gfCNCPoint3[9678] = {X 502.6885, Y 49.3200, Z -3.8333, A 0.000, B 0.000, C 0.000 }
gfCNCPoint3[9679] = {X 496.2450, Y 49.3200, Z -3.8333, A 0.000, B 0.000, C 0.000 }
gfCNCPoint3[9680] = {X 495.2885, Y 49.2128, Z -3.8333, A 0.000, B 0.000, C 0.000 }
gfCNCPoint3[9681] = {X 494.3794, Y 48.8964, Z -3.8333, A 0.000, B 0.000, C 0.000 }
gfCNCPoint3[9682] = {X 493.5630, Y 48.3866, Z -3.8333, A 0.000, B 0.000, C 0.000 }
gfCNCPoint3[9683] = {X 492.8797, Y 47.7087, Z -3.8333, A 0.000, B 0.000, C 0.000 }
gfCNCPoint3[9684] = {X 492.3635, Y 46.8963, Z -3.8333, A 0.000, B 0.000, C 0.000 }
gfCNCPoint3[9685] = {X 492.0399, Y 45.9898, Z -3.8333, A 0.000, B 0.000, C 0.000 }
gfCNCPoint3[9686] = {X 491.9252, Y 45.0341, Z -3.8333, A 0.000, B 0.000, C 0.000 }
gfCNCPoint3[9687] = {X 491.9254, Y 44.1494, Z -3.8333, A 0.000, B 0.000, C 0.000 }
gfCNCPoint3[9688] = {X 492.0359, Y 43.2364, Z -3.8333, A 0.000, B 0.000, C 0.000 }
gfCNCPoint3[9689] = {X 492.3371, Y 42.3675, Z -3.8333, A 0.000, B 0.000, C 0.000 }
gfCNCPoint3[9690] = {X 492.8153, Y 41.5821, Z -3.8333, A 0.000, B 0.000, C 0.000 }
gfCNCPoint3[9691] = {X 493.4490, Y 40.9157, Z -3.8333, A 0.000, B 0.000, C 0.000 }
gfCNCPoint3[9692] = {X 493.4490, Y 34.4738, Z -3.8333, A 0.000, B 0.000, C 0.000 }
gfCNCPoint3[9693] = {X 490.7241, Y 34.4738, Z -3.8333, A 0.000, B 0.000, C 0.000 }
gfCNCPoint3[9694] = {X 486.4400, Y 42.8164, Z -3.8333, A 0.000, B 0.000, C 0.000 }
gfCNCPoint3[9695] = {X 486.4449, Y 42.8296, Z -3.8333, A 0.000, B 0.000, C 0.000 }
gfCNCPoint3[9696] = {X 486.6109, Y 43.4908, Z -3.8333, A 0.000, B 0.000, C 0.000 }
gfCNCPoint3[9697] = {X 486.6708, Y 44.1699, Z -3.8333, A 0.000, B 0.000, C 0.000 }
gfCNCPoint3[9698] = {X 486.6710, Y 45.0000, Z -3.8333, A 0.000, B 0.000, C 0.000 }
gfCNCPoint3[9699] = {X 486.5627, Y 45.9613, Z -3.8333, A 0.000, B 0.000, C 0.000 }
gfCNCPoint3[9700] = {X 486.2432, Y 46.8744, Z -3.8333, A 0.000, B 0.000, C 0.000 }
gfCNCPoint3[9701] = {X 485.7285, Y 47.6935, Z -3.8333, A 0.000, B 0.000, C 0.000 }
gfCNCPoint3[9702] = {X 485.0445, Y 48.3775, Z -3.8333, A 0.000, B 0.000, C 0.000 }
gfCNCPoint3[9703] = {X 484.2254, Y 48.8922, Z -3.8333, A 0.000, B 0.000, C 0.000 }
gfCNCPoint3[9704] = {X 483.3123, Y 49.2117, Z -3.8333, A 0.000, B 0.000, C 0.000 }
gfCNCPoint3[9705] = {X 482.3510, Y 49.3200, Z -3.8333, A 0.000, B 0.000, C 0.000 }
gfCNCPoint3[9706] = {X 475.7650, Y 49.3200, Z -3.8333, A 0.000, B 0.000, C 0.000 }
gfCNCPoint3[9707] = {X 474.8037, Y 49.2117, Z -3.8333, A 0.000, B 0.000, C 0.000 }
gfCNCPoint3[9708] = {X 473.8906, Y 48.8922, Z -3.8333, A 0.000, B 0.000, C 0.000 }
gfCNCPoint3[9709] = {X 473.0715, Y 48.3775, Z -3.8333, A 0.000, B 0.000, C 0.000 }
gfCNCPoint3[9710] = {X 472.3875, Y 47.6935, Z -3.8333, A 0.000, B 0.000, C 0.000 }
gfCNCPoint3[9711] = {X 471.8728, Y 46.8745, Z -3.8333, A 0.000, B 0.000, C 0.000 }
gfCNCPoint3[9712] = {X 471.5533, Y 45.9614, Z -3.8333, A 0.000, B 0.000, C 0.000 }
gfCNCPoint3[9713] = {X 471.4450, Y 45.0001, Z -3.8333, A 0.000, B 0.000, C 0.000 }
gfCNCPoint3[9714] = {X 471.4454, Y 44.1494, Z -3.8333, A 0.000, B 0.000, C 0.000 }
gfCNCPoint3[9715] = {X 471.5430, Y 43.2935, Z -3.8333, A 0.000, B 0.000, C 0.000 }
gfCNCPoint3[9716] = {X 471.8086, Y 42.4740, Z -3.8333, A 0.000, B 0.000, C 0.000 }
gfCNCPoint3[9717] = {X 472.2314, Y 41.7236, Z -3.8333, A 0.000, B 0.000, C 0.000 }
gfCNCPoint3[9718] = {X 472.7947, Y 41.0719, Z -3.8333, A 0.000, B 0.000, C 0.000 }
gfCNCPoint3[9719] = {X 473.4762, Y 40.5449, Z -3.8333, A 0.000, B 0.000, C 0.000 }
gfCNCPoint3[9720] = {X 474.2486, Y 40.1637, Z -3.8333, A 0.000, B 0.000, C 0.000 }
gfCNCPoint3[9721] = {X 478.2331, Y 32.3645, Z -3.8333, A 0.000, B 0.000, C 0.000 }
gfCNCPoint3[9722] = {X 476.9697, Y 31.4968, Z -3.8333, A 0.000, B 0.000, C 0.000 }
gfCNCPoint3[9723] = {X 475.8333, Y 30.4684, Z -3.8333, A 0.000, B 0.000, C 0.000 }
gfCNCPoint3[9724] = {X 474.8441, Y 29.2977, Z -3.8333, A 0.000, B 0.000, C 0.000 }
gfCNCPoint3[9725] = {X 474.0198, Y 28.0056, Z -3.8333, A 0.000, B 0.000, C 0.000 }
gfCNCPoint3[9726] = {X 473.3752, Y 26.6150, Z -3.8333, A 0.000, B 0.000, C 0.000 }
gfCNCPoint3[9727] = {X 472.9218, Y 25.1510, Z -3.8333, A 0.000, B 0.000, C 0.000 }
gfCNCPoint3[9728] = {X 472.6083, Y 23.4679, Z -3.8333, A 0.000, B 0.000, C 0.000 }
gfCNCPoint3[9729] = {X 472.4682, Y 21.7616, Z -3.8333, A 0.000, B 0.000, C 0.000 }
gfCNCPoint3[9730] = {X 472.5029, Y 20.0499, Z -3.8333, A 0.000, B 0.000, C 0.000 }
gfCNCPoint3[9731] = {X 472.7121, Y 18.3506, Z -3.8333, A 0.000, B 0.000, C 0.000 }
gfCNCPoint3[9732] = {X 473.0935, Y 16.6816, Z -3.8333, A 0.000, B 0.000, C 0.000 }
gfCNCPoint3[9733] = {X 473.6361, Y 15.1667, Z -3.8333, A 0.000, B 0.000, C 0.000 }
gfCNCPoint3[9734] = {X 474.3793, Y 13.7395, Z -3.8333, A 0.000, B 0.000, C 0.000 }
gfCNCPoint3[9735] = {X 475.3094, Y 12.4264, Z -3.8333, A 0.000, B 0.000, C 0.000 }
gfCNCPoint3[9736] = {X 476.4090, Y 11.2517, Z -3.8333, A 0.000, B 0.000, C 0.000 }
gfCNCPoint3[9737] = {X 477.6579, Y 10.2370, Z -3.8333, A 0.000, B 0.000, C 0.000 }
gfCNCPoint3[9738] = {X 479.0330, Y 9.4012, Z -3.8333, A 0.000, B 0.000, C 0.000 }
gfCNCPoint3[9739] = {X 480.5087, Y 8.7598, Z -3.8333, A 0.000, B 0.000, C 0.000 }
gfCNCPoint3[9740] = {X 482.0579, Y 8.3246, Z -3.8333, A 0.000, B 0.000, C 0.000 }
gfCNCPoint3[9741] = {X 484.1552, Y 7.9976, Z -3.8333, A 0.000, B 0.000, C 0.000 }
gfCNCPoint3[9742] = {X 486.2747, Y 7.8831, Z -3.8333, A 0.000, B 0.000, C 0.000 }
gfCNCPoint3[9743] = {X 486.9679, Y 7.8709, Z -3.8333, A 0.000, B 0.000, C 0.000 }
gfCNCPoint3[9744] = {X 492.3835, Y 7.8709, Z -3.8333, A 0.000, B 0.000, C 0.000 }
gfCNCPoint3[9745] = {X 492.3835, Y 3.8709, Z -3.8333, A 0.000, B 0.000, C 0.000 }
gfCNCPoint3[9746] = {X 492.3835, Y 7.9509, Z -3.8333, A 0.000, B 0.000, C 0.000 }
gfCNCPoint3[9747] = {X 502.2063, Y 7.9509, Z -3.8333, A 0.000, B 0.000, C 0.000 }
gfCNCPoint3[9748] = {X 502.7388, Y 7.9551, Z -3.8333, A 0.000, B 0.000, C 0.000 }
gfCNCPoint3[9749] = {X 503.6730, Y 8.0672, Z -3.8333, A 0.000, B 0.000, C 0.000 }
gfCNCPoint3[9750] = {X 504.5591, Y 8.3834, Z -3.8333, A 0.000, B 0.000, C 0.000 }
gfCNCPoint3[9751] = {X 505.3533, Y 8.8880, Z -3.8333, A 0.000, B 0.000, C 0.000 }
gfCNCPoint3[9752] = {X 506.0160, Y 9.5559, Z -3.8333, A 0.000, B 0.000, C 0.000 }
gfCNCPoint3[9753] = {X 506.5144, Y 10.3540, Z -3.8333, A 0.000, B 0.000, C 0.000 }
gfCNCPoint3[9754] = {X 506.8237, Y 11.2426, Z -3.8333, A 0.000, B 0.000, C 0.000 }
gfCNCPoint3[9755] = {X 506.9285, Y 12.1776, Z -3.8333, A 0.000, B 0.000, C 0.000 }
gfCNCPoint3[9756] = {X 506.9285, Y 12.9781, Z -3.8333, A 0.000, B 0.000, C 0.000 }
gfCNCPoint3[9757] = {X 506.8270, Y 13.9000, Z -3.8333, A 0.000, B 0.000, C 0.000 }
gfCNCPoint3[9758] = {X 506.5276, Y 14.7777, Z -3.8333, A 0.000, B 0.000, C 0.000 }
gfCNCPoint3[9759] = {X 506.0445, Y 15.5693, Z -3.8333, A 0.000, B 0.000, C 0.000 }
gfCNCPoint3[9760] = {X 505.4009, Y 16.2369, Z -3.8333, A 0.000, B 0.000, C 0.000 }
gfCNCPoint3[9761] = {X 505.4008, Y 40.9504, Z -3.8333, A 0.000, B 0.000, C 0.000 }
gfCNCPoint3[9762] = {X 505.4291, Y 40.9736, Z -3.8333, A 0.000, B 0.000, C 0.000 }
gfCNCPoint3[9763] = {X 506.0558, Y 41.6322, Z -3.8333, A 0.000, B 0.000, C 0.000 }
gfCNCPoint3[9764] = {X 506.5277, Y 42.4092, Z -3.8333, A 0.000, B 0.000, C 0.000 }
gfCNCPoint3[9765] = {X 506.8230, Y 43.2690, Z -3.8333, A 0.000, B 0.000, C 0.000 }
gfCNCPoint3[9766] = {X 506.9283, Y 44.1720, Z -3.8333, A 0.000, B 0.000, C 0.000 }
gfCNCPoint3[9767] = {X 506.9285, Y 45.0000, Z -3.8333, A 0.000, B 0.000, C 0.000 }
gfCNCPoint3[9768] = {X 506.8222, Y 45.9435, Z -3.8333, A 0.000, B 0.000, C 0.000 }
gfCNCPoint3[9769] = {X 506.5086, Y 46.8397, Z -3.8333, A 0.000, B 0.000, C 0.000 }
gfCNCPoint3[9770] = {X 506.0035, Y 47.6436, Z -3.8333, A 0.000, B 0.000, C 0.000 }
gfCNCPoint3[9771] = {X 505.3321, Y 48.3150, Z -3.8333, A 0.000, B 0.000, C 0.000 }
gfCNCPoint3[9772] = {X 504.5282, Y 48.8201, Z -3.8333, A 0.000, B 0.000, C 0.000 }
gfCNCPoint3[9773] = {X 503.6320, Y 49.1337, Z -3.8333, A 0.000, B 0.000, C 0.000 }
gfCNCPoint3[9774] = {X 502.6885, Y 49.2400, Z -3.8333, A 0.000, B 0.000, C 0.000 }
gfCNCPoint3[9775] = {X 496.2450, Y 49.2400, Z -3.8333, A 0.000, B 0.000, C 0.000 }
gfCNCPoint3[9776] = {X 495.3062, Y 49.1348, Z -3.8333, A 0.000, B 0.000, C 0.000 }
gfCNCPoint3[9777] = {X 494.4140, Y 48.8242, Z -3.8333, A 0.000, B 0.000, C 0.000 }
gfCNCPoint3[9778] = {X 493.6127, Y 48.3239, Z -3.8333, A 0.000, B 0.000, C 0.000 }
gfCNCPoint3[9779] = {X 492.9420, Y 47.6585, Z -3.8333, A 0.000, B 0.000, C 0.000 }
gfCNCPoint3[9780] = {X 492.4354, Y 46.8612, Z -3.8333, A 0.000, B 0.000, C 0.000 }
gfCNCPoint3[9781] = {X 492.1178, Y 45.9714, Z -3.8333, A 0.000, B 0.000, C 0.000 }
gfCNCPoint3[9782] = {X 492.0052, Y 45.0335, Z -3.8333, A 0.000, B 0.000, C 0.000 }
gfCNCPoint3[9783] = {X 492.0054, Y 44.1505, Z -3.8333, A 0.000, B 0.000, C 0.000 }
gfCNCPoint3[9784] = {X 492.1159, Y 43.2454, Z -3.8333, A 0.000, B 0.000, C 0.000 }
gfCNCPoint3[9785] = {X 492.4173, Y 42.3850, Z -3.8333, A 0.000, B 0.000, C 0.000 }
gfCNCPoint3[9786] = {X 492.8957, Y 41.6088, Z -3.8333, A 0.000, B 0.000, C 0.000 }
gfCNCPoint3[9787] = {X 493.5290, Y 40.9529, Z -3.8333, A 0.000, B 0.000, C 0.000 }
gfCNCPoint3[9788] = {X 493.5290, Y 34.3938, Z -3.8333, A 0.000, B 0.000, C 0.000 }
gfCNCPoint3[9789] = {X 490.6753, Y 34.3938, Z -3.8333, A 0.000, B 0.000, C 0.000 }
gfCNCPoint3[9790] = {X 486.3526, Y 42.8115, Z -3.8333, A 0.000, B 0.000, C 0.000 }
gfCNCPoint3[9791] = {X 486.3696, Y 42.8564, Z -3.8333, A 0.000, B 0.000, C 0.000 }
gfCNCPoint3[9792] = {X 486.5322, Y 43.5048, Z -3.8333, A 0.000, B 0.000, C 0.000 }
gfCNCPoint3[9793] = {X 486.5908, Y 44.1706, Z -3.8333, A 0.000, B 0.000, C 0.000 }
gfCNCPoint3[9794] = {X 486.5910, Y 45.0000, Z -3.8333, A 0.000, B 0.000, C 0.000 }
gfCNCPoint3[9795] = {X 486.4847, Y 45.9435, Z -3.8333, A 0.000, B 0.000, C 0.000 }
gfCNCPoint3[9796] = {X 486.1711, Y 46.8397, Z -3.8333, A 0.000, B 0.000, C 0.000 }
gfCNCPoint3[9797] = {X 485.6660, Y 47.6436, Z -3.8333, A 0.000, B 0.000, C 0.000 }
gfCNCPoint3[9798] = {X 484.9946, Y 48.3150, Z -3.8333, A 0.000, B 0.000, C 0.000 }
gfCNCPoint3[9799] = {X 484.1907, Y 48.8201, Z -3.8333, A 0.000, B 0.000, C 0.000 }
gfCNCPoint3[9800] = {X 483.2945, Y 49.1337, Z -3.8333, A 0.000, B 0.000, C 0.000 }
gfCNCPoint3[9801] = {X 482.3510, Y 49.2400, Z -3.8333, A 0.000, B 0.000, C 0.000 }
gfCNCPoint3[9802] = {X 475.7650, Y 49.2400, Z -3.8333, A 0.000, B 0.000, C 0.000 }
gfCNCPoint3[9803] = {X 474.8215, Y 49.1337, Z -3.8333, A 0.000, B 0.000, C 0.000 }
gfCNCPoint3[9804] = {X 473.9253, Y 48.8201, Z -3.8333, A 0.000, B 0.000, C 0.000 }
gfCNCPoint3[9805] = {X 473.1214, Y 48.3150, Z -3.8333, A 0.000, B 0.000, C 0.000 }
gfCNCPoint3[9806] = {X 472.4500, Y 47.6436, Z -3.8333, A 0.000, B 0.000, C 0.000 }
gfCNCPoint3[9807] = {X 471.9449, Y 46.8397, Z -3.8333, A 0.000, B 0.000, C 0.000 }
gfCNCPoint3[9808] = {X 471.6313, Y 45.9436, Z -3.8333, A 0.000, B 0.000, C 0.000 }
gfCNCPoint3[9809] = {X 471.5250, Y 45.0001, Z -3.8333, A 0.000, B 0.000, C 0.000 }
gfCNCPoint3[9810] = {X 471.5254, Y 44.1505, Z -3.8333, A 0.000, B 0.000, C 0.000 }
gfCNCPoint3[9811] = {X 471.6223, Y 43.3054, Z -3.8333, A 0.000, B 0.000, C 0.000 }
gfCNCPoint3[9812] = {X 471.8860, Y 42.4967, Z -3.8333, A 0.000, B 0.000, C 0.000 }
gfCNCPoint3[9813] = {X 472.3057, Y 41.7570, Z -3.8333, A 0.000, B 0.000, C 0.000 }
gfCNCPoint3[9814] = {X 472.8647, Y 41.1159, Z -3.8333, A 0.000, B 0.000, C 0.000 }
gfCNCPoint3[9815] = {X 473.5404, Y 40.5992, Z -3.8333, A 0.000, B 0.000, C 0.000 }
gfCNCPoint3[9816] = {X 474.3057, Y 40.2278, Z -3.8333, A 0.000, B 0.000, C 0.000 }
gfCNCPoint3[9817] = {X 478.3386, Y 32.3338, Z -3.8333, A 0.000, B 0.000, C 0.000 }
gfCNCPoint3[9818] = {X 477.0685, Y 31.4727, Z -3.8333, A 0.000, B 0.000, C 0.000 }
gfCNCPoint3[9819] = {X 475.9257, Y 30.4488, Z -3.8333, A 0.000, B 0.000, C 0.000 }
gfCNCPoint3[9820] = {X 474.9308, Y 29.2805, Z -3.8333, A 0.000, B 0.000, C 0.000 }
gfCNCPoint3[9821] = {X 474.1021, Y 27.9891, Z -3.8333, A 0.000, B 0.000, C 0.000 }
gfCNCPoint3[9822] = {X 473.4544, Y 26.5980, Z -3.8333, A 0.000, B 0.000, C 0.000 }
gfCNCPoint3[9823] = {X 472.9996, Y 25.1325, Z -3.8333, A 0.000, B 0.000, C 0.000 }
gfCNCPoint3[9824] = {X 472.6876, Y 23.4574, Z -3.8333, A 0.000, B 0.000, C 0.000 }
gfCNCPoint3[9825] = {X 472.5482, Y 21.7592, Z -3.8333, A 0.000, B 0.000, C 0.000 }
gfCNCPoint3[9826] = {X 472.5827, Y 20.0556, Z -3.8333, A 0.000, B 0.000, C 0.000 }
gfCNCPoint3[9827] = {X 472.7909, Y 18.3645, Z -3.8333, A 0.000, B 0.000, C 0.000 }
gfCNCPoint3[9828] = {X 473.1704, Y 16.7034, Z -3.8333, A 0.000, B 0.000, C 0.000 }
gfCNCPoint3[9829] = {X 473.7094, Y 15.1988, Z -3.8333, A 0.000, B 0.000, C 0.000 }
gfCNCPoint3[9830] = {X 474.4476, Y 13.7812, Z -3.8333, A 0.000, B 0.000, C 0.000 }
gfCNCPoint3[9831] = {X 475.3714, Y 12.4770, Z -3.8333, A 0.000, B 0.000, C 0.000 }
gfCNCPoint3[9832] = {X 476.4636, Y 11.3102, Z -3.8333, A 0.000, B 0.000, C 0.000 }
gfCNCPoint3[9833] = {X 477.7040, Y 10.3024, Z -3.8333, A 0.000, B 0.000, C 0.000 }
gfCNCPoint3[9834] = {X 479.0698, Y 9.4722, Z -3.8333, A 0.000, B 0.000, C 0.000 }
gfCNCPoint3[9835] = {X 480.5356, Y 8.8351, Z -3.8333, A 0.000, B 0.000, C 0.000 }
gfCNCPoint3[9836] = {X 482.0742, Y 8.4029, Z -3.8333, A 0.000, B 0.000, C 0.000 }
gfCNCPoint3[9837] = {X 484.1638, Y 8.0772, Z -3.8333, A 0.000, B 0.000, C 0.000 }
gfCNCPoint3[9838] = {X 486.2756, Y 7.9631, Z -3.8333, A 0.000, B 0.000, C 0.000 }
gfCNCPoint3[9839] = {X 486.9686, Y 7.9509, Z -3.8333, A 0.000, B 0.000, C 0.000 }
gfCNCPoint3[9840] = {X 492.3835, Y 7.9509, Z -3.8333, A 0.000, B 0.000, C 0.000 }
gfCNCPoint3[9841] = {X 492.3835, Y 3.9509, Z -3.8333, A 0.000, B 0.000, C 0.000 }
gfCNCPoint3[9842] = {X 492.3835, Y 8.0309, Z -3.8333, A 0.000, B 0.000, C 0.000 }
gfCNCPoint3[9843] = {X 502.2059, Y 8.0309, Z -3.8333, A 0.000, B 0.000, C 0.000 }
gfCNCPoint3[9844] = {X 502.7381, Y 8.0351, Z -3.8333, A 0.000, B 0.000, C 0.000 }
gfCNCPoint3[9845] = {X 503.6546, Y 8.1451, Z -3.8333, A 0.000, B 0.000, C 0.000 }
gfCNCPoint3[9846] = {X 504.5240, Y 8.4553, Z -3.8333, A 0.000, B 0.000, C 0.000 }
gfCNCPoint3[9847] = {X 505.3031, Y 8.9503, Z -3.8333, A 0.000, B 0.000, C 0.000 }
gfCNCPoint3[9848] = {X 505.9533, Y 9.6056, Z -3.8333, A 0.000, B 0.000, C 0.000 }
gfCNCPoint3[9849] = {X 506.4422, Y 10.3885, Z -3.8333, A 0.000, B 0.000, C 0.000 }
gfCNCPoint3[9850] = {X 506.7457, Y 11.2603, Z -3.8333, A 0.000, B 0.000, C 0.000 }
gfCNCPoint3[9851] = {X 506.8485, Y 12.1776, Z -3.8333, A 0.000, B 0.000, C 0.000 }
gfCNCPoint3[9852] = {X 506.8485, Y 12.9781, Z -3.8333, A 0.000, B 0.000, C 0.000 }
gfCNCPoint3[9853] = {X 506.7469, Y 13.8917, Z -3.8333, A 0.000, B 0.000, C 0.000 }
gfCNCPoint3[9854] = {X 506.4472, Y 14.7606, Z -3.8333, A 0.000, B 0.000, C 0.000 }
gfCNCPoint3[9855] = {X 505.9640, Y 15.5425, Z -3.8333, A 0.000, B 0.000, C 0.000 }
gfCNCPoint3[9856] = {X 505.3209, Y 16.1992, Z -3.8333, A 0.000, B 0.000, C 0.000 }
gfCNCPoint3[9857] = {X 505.3208, Y 40.9888, Z -3.8333, A 0.000, B 0.000, C 0.000 }
gfCNCPoint3[9858] = {X 505.3677, Y 41.0265, Z -3.8333, A 0.000, B 0.000, C 0.000 }
gfCNCPoint3[9859] = {X 505.9865, Y 41.6733, Z -3.8333, A 0.000, B 0.000, C 0.000 }
gfCNCPoint3[9860] = {X 506.4525, Y 42.4375, Z -3.8333, A 0.000, B 0.000, C 0.000 }
gfCNCPoint3[9861] = {X 506.7443, Y 43.2837, Z -3.8333, A 0.000, B 0.000, C 0.000 }
gfCNCPoint3[9862] = {X 506.8483, Y 44.1727, Z -3.8333, A 0.000, B 0.000, C 0.000 }
gfCNCPoint3[9863] = {X 506.8485, Y 45.0000, Z -3.8333, A 0.000, B 0.000, C 0.000 }
gfCNCPoint3[9864] = {X 506.7442, Y 45.9257, Z -3.8333, A 0.000, B 0.000, C 0.000 }
gfCNCPoint3[9865] = {X 506.4365, Y 46.8050, Z -3.8333, A 0.000, B 0.000, C 0.000 }
gfCNCPoint3[9866] = {X 505.9409, Y 47.5937, Z -3.8333, A 0.000, B 0.000, C 0.000 }
gfCNCPoint3[9867] = {X 505.2822, Y 48.2524, Z -3.8333, A 0.000, B 0.000, C 0.000 }
gfCNCPoint3[9868] = {X 504.4934, Y 48.7480, Z -3.8333, A 0.000, B 0.000, C 0.000 }
gfCNCPoint3[9869] = {X 503.6142, Y 49.0557, Z -3.8333, A 0.000, B 0.000, C 0.000 }
gfCNCPoint3[9870] = {X 502.6885, Y 49.1600, Z -3.8333, A 0.000, B 0.000, C 0.000 }
gfCNCPoint3[9871] = {X 496.2450, Y 49.1600, Z -3.8333, A 0.000, B 0.000, C 0.000 }
gfCNCPoint3[9872] = {X 495.3239, Y 49.0567, Z -3.8333, A 0.000, B 0.000, C 0.000 }
gfCNCPoint3[9873] = {X 494.4485, Y 48.7521, Z -3.8333, A 0.000, B 0.000, C 0.000 }
gfCNCPoint3[9874] = {X 493.6623, Y 48.2612, Z -3.8333, A 0.000, B 0.000, C 0.000 }
gfCNCPoint3[9875] = {X 493.0043, Y 47.6084, Z -3.8333, A 0.000, B 0.000, C 0.000 }
gfCNCPoint3[9876] = {X 492.5072, Y 46.8261, Z -3.8333, A 0.000, B 0.000, C 0.000 }
gfCNCPoint3[9877] = {X 492.1957, Y 45.9531, Z -3.8333, A 0.000, B 0.000, C 0.000 }
gfCNCPoint3[9878] = {X 492.0852, Y 45.0328, Z -3.8333, A 0.000, B 0.000, C 0.000 }
gfCNCPoint3[9879] = {X 492.0854, Y 44.1516, Z -3.8333, A 0.000, B 0.000, C 0.000 }
gfCNCPoint3[9880] = {X 492.1960, Y 43.2545, Z -3.8333, A 0.000, B 0.000, C 0.000 }
gfCNCPoint3[9881] = {X 492.4976, Y 42.4026, Z -3.8333, A 0.000, B 0.000, C 0.000 }
gfCNCPoint3[9882] = {X 492.9762, Y 41.6358, Z -3.8333, A 0.000, B 0.000, C 0.000 }
gfCNCPoint3[9883] = {X 493.6090, Y 40.9906, Z -3.8333, A 0.000, B 0.000, C 0.000 }
gfCNCPoint3[9884] = {X 493.6090, Y 34.3138, Z -3.8333, A 0.000, B 0.000, C 0.000 }
gfCNCPoint3[9885] = {X 490.6264, Y 34.3138, Z -3.8333, A 0.000, B 0.000, C 0.000 }
gfCNCPoint3[9886] = {X 486.2652, Y 42.8065, Z -3.8333, A 0.000, B 0.000, C 0.000 }
gfCNCPoint3[9887] = {X 486.2942, Y 42.8833, Z -3.8333, A 0.000, B 0.000, C 0.000 }
gfCNCPoint3[9888] = {X 486.4534, Y 43.5188, Z -3.8333, A 0.000, B 0.000, C 0.000 }
gfCNCPoint3[9889] = {X 486.5108, Y 44.1713, Z -3.8333, A 0.000, B 0.000, C 0.000 }
gfCNCPoint3[9890] = {X 486.5110, Y 45.0000, Z -3.8333, A 0.000, B 0.000, C 0.000 }
gfCNCPoint3[9891] = {X 486.4067, Y 45.9257, Z -3.8333, A 0.000, B 0.000, C 0.000 }
gfCNCPoint3[9892] = {X 486.0990, Y 46.8050, Z -3.8333, A 0.000, B 0.000, C 0.000 }
gfCNCPoint3[9893] = {X 485.6034, Y 47.5937, Z -3.8333, A 0.000, B 0.000, C 0.000 }
gfCNCPoint3[9894] = {X 484.9447, Y 48.2524, Z -3.8333, A 0.000, B 0.000, C 0.000 }
gfCNCPoint3[9895] = {X 484.1560, Y 48.7480, Z -3.8333, A 0.000, B 0.000, C 0.000 }
gfCNCPoint3[9896] = {X 483.2767, Y 49.0557, Z -3.8333, A 0.000, B 0.000, C 0.000 }
gfCNCPoint3[9897] = {X 482.3510, Y 49.1600, Z -3.8333, A 0.000, B 0.000, C 0.000 }
gfCNCPoint3[9898] = {X 475.7650, Y 49.1600, Z -3.8333, A 0.000, B 0.000, C 0.000 }
gfCNCPoint3[9899] = {X 474.8393, Y 49.0557, Z -3.8333, A 0.000, B 0.000, C 0.000 }
gfCNCPoint3[9900] = {X 473.9600, Y 48.7480, Z -3.8333, A 0.000, B 0.000, C 0.000 }
gfCNCPoint3[9901] = {X 473.1713, Y 48.2524, Z -3.8333, A 0.000, B 0.000, C 0.000 }
gfCNCPoint3[9902] = {X 472.5126, Y 47.5937, Z -3.8333, A 0.000, B 0.000, C 0.000 }
gfCNCPoint3[9903] = {X 472.0169, Y 46.8050, Z -3.8333, A 0.000, B 0.000, C 0.000 }
gfCNCPoint3[9904] = {X 471.7093, Y 45.9257, Z -3.8333, A 0.000, B 0.000, C 0.000 }
gfCNCPoint3[9905] = {X 471.6050, Y 45.0000, Z -3.8333, A 0.000, B 0.000, C 0.000 }
gfCNCPoint3[9906] = {X 471.6054, Y 44.1516, Z -3.8333, A 0.000, B 0.000, C 0.000 }
gfCNCPoint3[9907] = {X 471.7016, Y 43.3174, Z -3.8333, A 0.000, B 0.000, C 0.000 }
gfCNCPoint3[9908] = {X 471.9634, Y 42.5195, Z -3.8333, A 0.000, B 0.000, C 0.000 }
gfCNCPoint3[9909] = {X 472.3801, Y 41.7905, Z -3.8333, A 0.000, B 0.000, C 0.000 }
gfCNCPoint3[9910] = {X 472.9347, Y 41.1600, Z -3.8333, A 0.000, B 0.000, C 0.000 }
gfCNCPoint3[9911] = {X 473.6046, Y 40.6537, Z -3.8333, A 0.000, B 0.000, C 0.000 }
gfCNCPoint3[9912] = {X 474.3626, Y 40.2923, Z -3.8333, A 0.000, B 0.000, C 0.000 }
gfCNCPoint3[9913] = {X 478.4444, Y 32.3026, Z -3.8333, A 0.000, B 0.000, C 0.000 }
gfCNCPoint3[9914] = {X 477.1675, Y 31.4483, Z -3.8333, A 0.000, B 0.000, C 0.000 }
gfCNCPoint3[9915] = {X 476.0182, Y 30.4289, Z -3.8333, A 0.000, B 0.000, C 0.000 }
gfCNCPoint3[9916] = {X 475.0176, Y 29.2631, Z -3.8333, A 0.000, B 0.000, C 0.000 }
gfCNCPoint3[9917] = {X 474.1843, Y 27.9725, Z -3.8333, A 0.000, B 0.000, C 0.000 }
gfCNCPoint3[9918] = {X 473.5335, Y 26.5808, Z -3.8333, A 0.000, B 0.000, C 0.000 }
gfCNCPoint3[9919] = {X 473.0774, Y 25.1138, Z -3.8333, A 0.000, B 0.000, C 0.000 }
gfCNCPoint3[9920] = {X 472.7669, Y 23.4468, Z -3.8333, A 0.000, B 0.000, C 0.000 }
gfCNCPoint3[9921] = {X 472.6281, Y 21.7567, Z -3.8333, A 0.000, B 0.000, C 0.000 }
gfCNCPoint3[9922] = {X 472.6625, Y 20.0613, Z -3.8333, A 0.000, B 0.000, C 0.000 }
gfCNCPoint3[9923] = {X 472.8696, Y 18.3783, Z -3.8333, A 0.000, B 0.000, C 0.000 }
gfCNCPoint3[9924] = {X 473.2474, Y 16.7252, Z -3.8333, A 0.000, B 0.000, C 0.000 }
gfCNCPoint3[9925] = {X 473.7827, Y 15.2308, Z -3.8333, A 0.000, B 0.000, C 0.000 }
gfCNCPoint3[9926] = {X 474.5159, Y 13.8229, Z -3.8333, A 0.000, B 0.000, C 0.000 }
gfCNCPoint3[9927] = {X 475.4334, Y 12.5275, Z -3.8333, A 0.000, B 0.000, C 0.000 }
gfCNCPoint3[9928] = {X 476.5181, Y 11.3687, Z -3.8333, A 0.000, B 0.000, C 0.000 }
gfCNCPoint3[9929] = {X 477.7502, Y 10.3677, Z -3.8333, A 0.000, B 0.000, C 0.000 }
gfCNCPoint3[9930] = {X 479.1066, Y 9.5433, Z -3.8333, A 0.000, B 0.000, C 0.000 }
gfCNCPoint3[9931] = {X 480.5624, Y 8.9105, Z -3.8333, A 0.000, B 0.000, C 0.000 }
gfCNCPoint3[9932] = {X 482.0906, Y 8.4812, Z -3.8333, A 0.000, B 0.000, C 0.000 }
gfCNCPoint3[9933] = {X 484.1725, Y 8.1567, Z -3.8333, A 0.000, B 0.000, C 0.000 }
gfCNCPoint3[9934] = {X 486.2765, Y 8.0431, Z -3.8333, A 0.000, B 0.000, C 0.000 }
gfCNCPoint3[9935] = {X 486.9693, Y 8.0309, Z -3.8333, A 0.000, B 0.000, C 0.000 }
gfCNCPoint3[9936] = {X 492.3835, Y 8.0309, Z -3.8333, A 0.000, B 0.000, C 0.000 }
gfCNCPoint3[9937] = {X 492.3835, Y 4.0309, Z -3.8333, A 0.000, B 0.000, C 0.000 }
gfCNCPoint3[9938] = {X 492.3835, Y 8.1109, Z -3.8333, A 0.000, B 0.000, C 0.000 }
gfCNCPoint3[9939] = {X 502.2056, Y 8.1109, Z -3.8333, A 0.000, B 0.000, C 0.000 }
gfCNCPoint3[9940] = {X 502.7375, Y 8.1151, Z -3.8333, A 0.000, B 0.000, C 0.000 }
gfCNCPoint3[9941] = {X 503.6363, Y 8.2229, Z -3.8333, A 0.000, B 0.000, C 0.000 }
gfCNCPoint3[9942] = {X 504.4889, Y 8.5272, Z -3.8333, A 0.000, B 0.000, C 0.000 }
gfCNCPoint3[9943] = {X 505.2530, Y 9.0126, Z -3.8333, A 0.000, B 0.000, C 0.000 }
gfCNCPoint3[9944] = {X 505.8906, Y 9.6552, Z -3.8333, A 0.000, B 0.000, C 0.000 }
gfCNCPoint3[9945] = {X 506.3701, Y 10.4231, Z -3.8333, A 0.000, B 0.000, C 0.000 }
gfCNCPoint3[9946] = {X 506.6676, Y 11.2780, Z -3.8333, A 0.000, B 0.000, C 0.000 }
gfCNCPoint3[9947] = {X 506.7685, Y 12.1776, Z -3.8333, A 0.000, B 0.000, C 0.000 }
gfCNCPoint3[9948] = {X 506.7685, Y 12.9781, Z -3.8333, A 0.000, B 0.000, C 0.000 }
gfCNCPoint3[9949] = {X 506.6668, Y 13.8833, Z -3.8333, A 0.000, B 0.000, C 0.000 }
gfCNCPoint3[9950] = {X 506.3668, Y 14.7434, Z -3.8333, A 0.000, B 0.000, C 0.000 }
gfCNCPoint3[9951] = {X 505.8835, Y 15.5154, Z -3.8333, A 0.000, B 0.000, C 0.000 }
gfCNCPoint3[9952] = {X 505.2409, Y 16.1610, Z -3.8333, A 0.000, B 0.000, C 0.000 }
gfCNCPoint3[9953] = {X 505.2408, Y 41.0272, Z -3.8333, A 0.000, B 0.000, C 0.000 }
gfCNCPoint3[9954] = {X 505.3177, Y 41.0889, Z -3.8333, A 0.000, B 0.000, C 0.000 }
gfCNCPoint3[9955] = {X 505.9239, Y 41.7232, Z -3.8333, A 0.000, B 0.000, C 0.000 }
gfCNCPoint3[9956] = {X 506.3805, Y 42.4724, Z -3.8333, A 0.000, B 0.000, C 0.000 }
gfCNCPoint3[9957] = {X 506.6664, Y 43.3019, Z -3.8333, A 0.000, B 0.000, C 0.000 }
gfCNCPoint3[9958] = {X 506.7683, Y 44.1734, Z -3.8333, A 0.000, B 0.000, C 0.000 }
gfCNCPoint3[9959] = {X 506.7685, Y 45.0000, Z -3.8333, A 0.000, B 0.000, C 0.000 }
gfCNCPoint3[9960] = {X 506.6662, Y 45.9079, Z -3.8333, A 0.000, B 0.000, C 0.000 }
gfCNCPoint3[9961] = {X 506.3644, Y 46.7702, Z -3.8333, A 0.000, B 0.000, C 0.000 }
gfCNCPoint3[9962] = {X 505.8784, Y 47.5438, Z -3.8333, A 0.000, B 0.000, C 0.000 }
gfCNCPoint3[9963] = {X 505.2323, Y 48.1899, Z -3.8333, A 0.000, B 0.000, C 0.000 }
gfCNCPoint3[9964] = {X 504.4587, Y 48.6760, Z -3.8333, A 0.000, B 0.000, C 0.000 }
gfCNCPoint3[9965] = {X 503.5964, Y 48.9777, Z -3.8333, A 0.000, B 0.000, C 0.000 }
gfCNCPoint3[9966] = {X 502.6885, Y 49.0800, Z -3.8333, A 0.000, B 0.000, C 0.000 }
gfCNCPoint3[9967] = {X 496.2450, Y 49.0800, Z -3.8333, A 0.000, B 0.000, C 0.000 }
gfCNCPoint3[9968] = {X 495.3416, Y 48.9787, Z -3.8333, A 0.000, B 0.000, C 0.000 }
gfCNCPoint3[9969] = {X 494.4831, Y 48.6799, Z -3.8333, A 0.000, B 0.000, C 0.000 }
gfCNCPoint3[9970] = {X 493.7120, Y 48.1985, Z -3.8333, A 0.000, B 0.000, C 0.000 }
gfCNCPoint3[9971] = {X 493.0667, Y 47.5582, Z -3.8333, A 0.000, B 0.000, C 0.000 }
gfCNCPoint3[9972] = {X 492.5791, Y 46.7909, Z -3.8333, A 0.000, B 0.000, C 0.000 }
gfCNCPoint3[9973] = {X 492.2736, Y 45.9348, Z -3.8333, A 0.000, B 0.000, C 0.000 }
gfCNCPoint3[9974] = {X 492.1652, Y 45.0322, Z -3.8333, A 0.000, B 0.000, C 0.000 }
gfCNCPoint3[9975] = {X 492.1654, Y 44.1527, Z -3.8333, A 0.000, B 0.000, C 0.000 }
gfCNCPoint3[9976] = {X 492.2760, Y 43.2637, Z -3.8333, A 0.000, B 0.000, C 0.000 }
gfCNCPoint3[9977] = {X 492.5779, Y 42.4203, Z -3.8333, A 0.000, B 0.000, C 0.000 }
gfCNCPoint3[9978] = {X 493.0566, Y 41.6631, Z -3.8333, A 0.000, B 0.000, C 0.000 }
gfCNCPoint3[9979] = {X 493.6890, Y 41.0287, Z -3.8333, A 0.000, B 0.000, C 0.000 }
gfCNCPoint3[9980] = {X 493.6890, Y 34.2338, Z -3.8333, A 0.000, B 0.000, C 0.000 }
gfCNCPoint3[9981] = {X 490.5776, Y 34.2338, Z -3.8333, A 0.000, B 0.000, C 0.000 }
gfCNCPoint3[9982] = {X 486.1778, Y 42.8015, Z -3.8333, A 0.000, B 0.000, C 0.000 }
gfCNCPoint3[9983] = {X 486.2188, Y 42.9102, Z -3.8333, A 0.000, B 0.000, C 0.000 }
gfCNCPoint3[9984] = {X 486.3746, Y 43.5328, Z -3.8333, A 0.000, B 0.000, C 0.000 }
gfCNCPoint3[9985] = {X 486.4309, Y 44.1720, Z -3.8333, A 0.000, B 0.000, C 0.000 }
gfCNCPoint3[9986] = {X 486.4310, Y 45.0000, Z -3.8333, A 0.000, B 0.000, C 0.000 }
gfCNCPoint3[9987] = {X 486.3287, Y 45.9079, Z -3.8333, A 0.000, B 0.000, C 0.000 }
gfCNCPoint3[9988] = {X 486.0270, Y 46.7702, Z -3.8333, A 0.000, B 0.000, C 0.000 }
gfCNCPoint3[9989] = {X 485.5409, Y 47.5438, Z -3.8333, A 0.000, B 0.000, C 0.000 }
gfCNCPoint3[9990] = {X 484.8949, Y 48.1899, Z -3.8333, A 0.000, B 0.000, C 0.000 }
gfCNCPoint3[9991] = {X 484.1213, Y 48.6760, Z -3.8333, A 0.000, B 0.000, C 0.000 }
gfCNCPoint3[9992] = {X 483.2589, Y 48.9777, Z -3.8333, A 0.000, B 0.000, C 0.000 }
gfCNCPoint3[9993] = {X 482.3510, Y 49.0800, Z -3.8333, A 0.000, B 0.000, C 0.000 }
gfCNCPoint3[9994] = {X 475.7650, Y 49.0800, Z -3.8333, A 0.000, B 0.000, C 0.000 }
gfCNCPoint3[9995] = {X 474.8571, Y 48.9777, Z -3.8333, A 0.000, B 0.000, C 0.000 }
gfCNCPoint3[9996] = {X 473.9947, Y 48.6760, Z -3.8333, A 0.000, B 0.000, C 0.000 }
gfCNCPoint3[9997] = {X 473.2211, Y 48.1899, Z -3.8333, A 0.000, B 0.000, C 0.000 }
gfCNCPoint3[9998] = {X 472.5751, Y 47.5438, Z -3.8333, A 0.000, B 0.000, C 0.000 }
gfCNCPoint3[9999] = {X 472.0890, Y 46.7702, Z -3.8333, A 0.000, B 0.000, C 0.000 }
gfCNCPoint3[10000] = {X 471.7873, Y 45.9079, Z -3.8333, A 0.000, B 0.000, C 0.000 }
gfCNCPoint3[10001] = {X 471.6850, Y 45.0000, Z -3.8333, A 0.000, B 0.000, C 0.000 }
gfCNCPoint3[10002] = {X 471.6853, Y 44.1527, Z -3.8333, A 0.000, B 0.000, C 0.000 }
gfCNCPoint3[10003] = {X 471.7809, Y 43.3294, Z -3.8333, A 0.000, B 0.000, C 0.000 }
gfCNCPoint3[10004] = {X 472.0408, Y 42.5424, Z -3.8333, A 0.000, B 0.000, C 0.000 }
gfCNCPoint3[10005] = {X 472.4544, Y 41.8242, Z -3.8333, A 0.000, B 0.000, C 0.000 }
gfCNCPoint3[10006] = {X 473.0046, Y 41.2044, Z -3.8333, A 0.000, B 0.000, C 0.000 }
gfCNCPoint3[10007] = {X 473.6687, Y 40.7085, Z -3.8333, A 0.000, B 0.000, C 0.000 }
gfCNCPoint3[10008] = {X 474.4193, Y 40.3571, Z -3.8333, A 0.000, B 0.000, C 0.000 }
gfCNCPoint3[10009] = {X 478.5504, Y 32.2710, Z -3.8333, A 0.000, B 0.000, C 0.000 }
gfCNCPoint3[10010] = {X 477.2667, Y 31.4236, Z -3.8333, A 0.000, B 0.000, C 0.000 }
gfCNCPoint3[10011] = {X 476.1109, Y 30.4089, Z -3.8333, A 0.000, B 0.000, C 0.000 }
gfCNCPoint3[10012] = {X 475.1045, Y 29.2457, Z -3.8333, A 0.000, B 0.000, C 0.000 }
gfCNCPoint3[10013] = {X 474.2665, Y 27.9559, Z -3.8333, A 0.000, B 0.000, C 0.000 }
gfCNCPoint3[10014] = {X 473.6127, Y 26.5637, Z -3.8333, A 0.000, B 0.000, C 0.000 }
gfCNCPoint3[10015] = {X 473.1552, Y 25.0952, Z -3.8333, A 0.000, B 0.000, C 0.000 }
gfCNCPoint3[10016] = {X 472.8462, Y 23.4362, Z -3.8333, A 0.000, B 0.000, C 0.000 }
gfCNCPoint3[10017] = {X 472.7081, Y 21.7543, Z -3.8333, A 0.000, B 0.000, C 0.000 }
gfCNCPoint3[10018] = {X 472.7423, Y 20.0670, Z -3.8333, A 0.000, B 0.000, C 0.000 }
gfCNCPoint3[10019] = {X 472.9484, Y 18.3921, Z -3.8333, A 0.000, B 0.000, C 0.000 }
gfCNCPoint3[10020] = {X 473.3244, Y 16.7470, Z -3.8333, A 0.000, B 0.000, C 0.000 }
gfCNCPoint3[10021] = {X 473.8560, Y 15.2628, Z -3.8333, A 0.000, B 0.000, C 0.000 }
gfCNCPoint3[10022] = {X 474.5842, Y 13.8646, Z -3.8333, A 0.000, B 0.000, C 0.000 }
gfCNCPoint3[10023] = {X 475.4954, Y 12.5781, Z -3.8333, A 0.000, B 0.000, C 0.000 }
gfCNCPoint3[10024] = {X 476.5727, Y 11.4272, Z -3.8333, A 0.000, B 0.000, C 0.000 }
gfCNCPoint3[10025] = {X 477.7963, Y 10.4331, Z -3.8333, A 0.000, B 0.000, C 0.000 }
gfCNCPoint3[10026] = {X 479.1434, Y 9.6143, Z -3.8333, A 0.000, B 0.000, C 0.000 }
gfCNCPoint3[10027] = {X 480.5892, Y 8.9859, Z -3.8333, A 0.000, B 0.000, C 0.000 }
gfCNCPoint3[10028] = {X 482.1069, Y 8.5595, Z -3.8333, A 0.000, B 0.000, C 0.000 }
gfCNCPoint3[10029] = {X 484.1811, Y 8.2362, Z -3.8333, A 0.000, B 0.000, C 0.000 }
gfCNCPoint3[10030] = {X 486.2773, Y 8.1231, Z -3.8333, A 0.000, B 0.000, C 0.000 }
gfCNCPoint3[10031] = {X 486.9700, Y 8.1109, Z -3.8333, A 0.000, B 0.000, C 0.000 }
gfCNCPoint3[10032] = {X 492.3835, Y 8.1109, Z -3.8333, A 0.000, B 0.000, C 0.000 }
gfCNCPoint3[10033] = {X 492.3835, Y 4.1109, Z -3.8333, A 0.000, B 0.000, C 0.000 }
gfCNCPoint3[10034] = {X 492.3835, Y 8.1909, Z -3.8333, A 0.000, B 0.000, C 0.000 }
gfCNCPoint3[10035] = {X 502.2053, Y 8.1909, Z -3.8333, A 0.000, B 0.000, C 0.000 }
gfCNCPoint3[10036] = {X 502.7369, Y 8.1951, Z -3.8333, A 0.000, B 0.000, C 0.000 }
gfCNCPoint3[10037] = {X 503.6180, Y 8.3008, Z -3.8333, A 0.000, B 0.000, C 0.000 }
gfCNCPoint3[10038] = {X 504.4538, Y 8.5990, Z -3.8333, A 0.000, B 0.000, C 0.000 }
gfCNCPoint3[10039] = {X 505.2028, Y 9.0749, Z -3.8333, A 0.000, B 0.000, C 0.000 }
gfCNCPoint3[10040] = {X 505.8279, Y 9.7049, Z -3.8333, A 0.000, B 0.000, C 0.000 }
gfCNCPoint3[10041] = {X 506.2979, Y 10.4576, Z -3.8333, A 0.000, B 0.000, C 0.000 }
gfCNCPoint3[10042] = {X 506.5896, Y 11.2957, Z -3.8333, A 0.000, B 0.000, C 0.000 }
gfCNCPoint3[10043] = {X 506.6885, Y 12.1776, Z -3.8333, A 0.000, B 0.000, C 0.000 }
gfCNCPoint3[10044] = {X 506.6883, Y 13.0192, Z -3.8333, A 0.000, B 0.000, C 0.000 }
gfCNCPoint3[10045] = {X 506.5796, Y 13.9049, Z -3.8333, A 0.000, B 0.000, C 0.000 }
gfCNCPoint3[10046] = {X 506.2773, Y 14.7444, Z -3.8333, A 0.000, B 0.000, C 0.000 }
gfCNCPoint3[10047] = {X 505.7964, Y 15.4961, Z -3.8333, A 0.000, B 0.000, C 0.000 }
gfCNCPoint3[10048] = {X 505.1609, Y 16.1224, Z -3.8333, A 0.000, B 0.000, C 0.000 }
gfCNCPoint3[10049] = {X 505.1608, Y 41.0656, Z -3.8333, A 0.000, B 0.000, C 0.000 }
gfCNCPoint3[10050] = {X 505.2997, Y 41.1787, Z -3.8333, A 0.000, B 0.000, C 0.000 }
gfCNCPoint3[10051] = {X 505.8858, Y 41.8052, Z -3.8333, A 0.000, B 0.000, C 0.000 }
gfCNCPoint3[10052] = {X 506.3248, Y 42.5422, Z -3.8333, A 0.000, B 0.000, C 0.000 }
gfCNCPoint3[10053] = {X 506.5965, Y 43.3560, Z -3.8333, A 0.000, B 0.000, C 0.000 }
gfCNCPoint3[10054] = {X 506.6885, Y 44.2089, Z -3.8333, A 0.000, B 0.000, C 0.000 }
gfCNCPoint3[10055] = {X 506.6885, Y 45.0000, Z -3.8333, A 0.000, B 0.000, C 0.000 }
gfCNCPoint3[10056] = {X 506.5882, Y 45.8901, Z -3.8333, A 0.000, B 0.000, C 0.000 }
gfCNCPoint3[10057] = {X 506.2924, Y 46.7355, Z -3.8333, A 0.000, B 0.000, C 0.000 }
gfCNCPoint3[10058] = {X 505.8158, Y 47.4940, Z -3.8333, A 0.000, B 0.000, C 0.000 }
gfCNCPoint3[10059] = {X 505.1825, Y 48.1273, Z -3.8333, A 0.000, B 0.000, C 0.000 }
gfCNCPoint3[10060] = {X 504.4240, Y 48.6039, Z -3.8333, A 0.000, B 0.000, C 0.000 }
gfCNCPoint3[10061] = {X 503.5786, Y 48.8997, Z -3.8333, A 0.000, B 0.000, C 0.000 }
gfCNCPoint3[10062] = {X 502.6885, Y 49.0000, Z -3.8333, A 0.000, B 0.000, C 0.000 }
gfCNCPoint3[10063] = {X 496.2450, Y 49.0000, Z -3.8333, A 0.000, B 0.000, C 0.000 }
gfCNCPoint3[10064] = {X 495.3549, Y 48.8997, Z -3.8333, A 0.000, B 0.000, C 0.000 }
gfCNCPoint3[10065] = {X 494.5095, Y 48.6039, Z -3.8333, A 0.000, B 0.000, C 0.000 }
gfCNCPoint3[10066] = {X 493.7511, Y 48.1273, Z -3.8333, A 0.000, B 0.000, C 0.000 }
gfCNCPoint3[10067] = {X 493.1177, Y 47.4939, Z -3.8333, A 0.000, B 0.000, C 0.000 }
gfCNCPoint3[10068] = {X 492.6411, Y 46.7355, Z -3.8333, A 0.000, B 0.000, C 0.000 }
gfCNCPoint3[10069] = {X 492.3453, Y 45.8900, Z -3.8333, A 0.000, B 0.000, C 0.000 }
gfCNCPoint3[10070] = {X 492.2450, Y 45.0000, Z -3.8333, A 0.000, B 0.000, C 0.000 }
gfCNCPoint3[10071] = {X 492.2454, Y 44.1538, Z -3.8333, A 0.000, B 0.000, C 0.000 }
gfCNCPoint3[10072] = {X 492.3560, Y 43.2730, Z -3.8333, A 0.000, B 0.000, C 0.000 }
gfCNCPoint3[10073] = {X 492.6582, Y 42.4382, Z -3.8333, A 0.000, B 0.000, C 0.000 }
gfCNCPoint3[10074] = {X 493.1371, Y 41.6907, Z -3.8333, A 0.000, B 0.000, C 0.000 }
gfCNCPoint3[10075] = {X 493.7690, Y 41.0672, Z -3.8333, A 0.000, B 0.000, C 0.000 }
gfCNCPoint3[10076] = {X 493.7690, Y 34.1538, Z -3.8333, A 0.000, B 0.000, C 0.000 }
gfCNCPoint3[10077] = {X 490.7730, Y 34.1538, Z -3.8333, A 0.000, B 0.000, C 0.000 }
gfCNCPoint3[10078] = {X 490.5300, Y 34.1513, Z -3.8333, A 0.000, B 0.000, C 0.000 }
gfCNCPoint3[10079] = {X 486.0905, Y 42.7966, Z -3.8333, A 0.000, B 0.000, C 0.000 }
gfCNCPoint3[10080] = {X 486.1473, Y 42.9484, Z -3.8333, A 0.000, B 0.000, C 0.000 }
gfCNCPoint3[10081] = {X 486.2998, Y 43.5705, Z -3.8333, A 0.000, B 0.000, C 0.000 }
gfCNCPoint3[10082] = {X 486.3510, Y 44.2089, Z -3.8333, A 0.000, B 0.000, C 0.000 }
gfCNCPoint3[10083] = {X 486.3510, Y 45.0000, Z -3.8333, A 0.000, B 0.000, C 0.000 }
gfCNCPoint3[10084] = {X 486.2507, Y 45.8901, Z -3.8333, A 0.000, B 0.000, C 0.000 }
gfCNCPoint3[10085] = {X 485.9549, Y 46.7355, Z -3.8333, A 0.000, B 0.000, C 0.000 }
gfCNCPoint3[10086] = {X 485.4783, Y 47.4940, Z -3.8333, A 0.000, B 0.000, C 0.000 }
gfCNCPoint3[10087] = {X 484.8450, Y 48.1273, Z -3.8333, A 0.000, B 0.000, C 0.000 }
gfCNCPoint3[10088] = {X 484.0866, Y 48.6039, Z -3.8333, A 0.000, B 0.000, C 0.000 }
gfCNCPoint3[10089] = {X 483.2411, Y 48.8997, Z -3.8333, A 0.000, B 0.000, C 0.000 }
gfCNCPoint3[10090] = {X 482.3510, Y 49.0000, Z -3.8333, A 0.000, B 0.000, C 0.000 }
gfCNCPoint3[10091] = {X 475.7650, Y 49.0000, Z -3.8333, A 0.000, B 0.000, C 0.000 }
gfCNCPoint3[10092] = {X 474.8749, Y 48.8997, Z -3.8333, A 0.000, B 0.000, C 0.000 }
gfCNCPoint3[10093] = {X 474.0294, Y 48.6039, Z -3.8333, A 0.000, B 0.000, C 0.000 }
gfCNCPoint3[10094] = {X 473.2710, Y 48.1273, Z -3.8333, A 0.000, B 0.000, C 0.000 }
gfCNCPoint3[10095] = {X 472.6376, Y 47.4940, Z -3.8333, A 0.000, B 0.000, C 0.000 }
gfCNCPoint3[10096] = {X 472.1611, Y 46.7355, Z -3.8333, A 0.000, B 0.000, C 0.000 }
gfCNCPoint3[10097] = {X 471.8652, Y 45.8901, Z -3.8333, A 0.000, B 0.000, C 0.000 }
gfCNCPoint3[10098] = {X 471.7650, Y 45.0000, Z -3.8333, A 0.000, B 0.000, C 0.000 }
gfCNCPoint3[10099] = {X 471.7653, Y 44.1538, Z -3.8333, A 0.000, B 0.000, C 0.000 }
gfCNCPoint3[10100] = {X 471.8601, Y 43.3414, Z -3.8333, A 0.000, B 0.000, C 0.000 }
gfCNCPoint3[10101] = {X 472.1182, Y 42.5654, Z -3.8333, A 0.000, B 0.000, C 0.000 }
gfCNCPoint3[10102] = {X 472.5286, Y 41.8580, Z -3.8333, A 0.000, B 0.000, C 0.000 }
gfCNCPoint3[10103] = {X 473.0744, Y 41.2489, Z -3.8333, A 0.000, B 0.000, C 0.000 }
gfCNCPoint3[10104] = {X 473.7327, Y 40.7635, Z -3.8333, A 0.000, B 0.000, C 0.000 }
gfCNCPoint3[10105] = {X 474.4759, Y 40.4222, Z -3.8333, A 0.000, B 0.000, C 0.000 }
gfCNCPoint3[10106] = {X 478.6566, Y 32.2388, Z -3.8333, A 0.000, B 0.000, C 0.000 }
gfCNCPoint3[10107] = {X 477.3661, Y 31.3986, Z -3.8333, A 0.000, B 0.000, C 0.000 }
gfCNCPoint3[10108] = {X 476.2037, Y 30.3886, Z -3.8333, A 0.000, B 0.000, C 0.000 }
gfCNCPoint3[10109] = {X 475.1915, Y 29.2281, Z -3.8333, A 0.000, B 0.000, C 0.000 }
gfCNCPoint3[10110] = {X 474.3489, Y 27.9392, Z -3.8333, A 0.000, B 0.000, C 0.000 }
gfCNCPoint3[10111] = {X 473.6918, Y 26.5465, Z -3.8333, A 0.000, B 0.000, C 0.000 }
gfCNCPoint3[10112] = {X 473.2330, Y 25.0766, Z -3.8333, A 0.000, B 0.000, C 0.000 }
gfCNCPoint3[10113] = {X 472.9255, Y 23.4256, Z -3.8333, A 0.000, B 0.000, C 0.000 }
gfCNCPoint3[10114] = {X 472.7881, Y 21.7518, Z -3.8333, A 0.000, B 0.000, C 0.000 }
gfCNCPoint3[10115] = {X 472.8221, Y 20.0727, Z -3.8333, A 0.000, B 0.000, C 0.000 }
gfCNCPoint3[10116] = {X 473.0272, Y 18.4059, Z -3.8333, A 0.000, B 0.000, C 0.000 }
gfCNCPoint3[10117] = {X 473.4014, Y 16.7687, Z -3.8333, A 0.000, B 0.000, C 0.000 }
gfCNCPoint3[10118] = {X 473.9294, Y 15.2949, Z -3.8333, A 0.000, B 0.000, C 0.000 }
gfCNCPoint3[10119] = {X 474.6525, Y 13.9063, Z -3.8333, A 0.000, B 0.000, C 0.000 }
gfCNCPoint3[10120] = {X 475.5574, Y 12.6287, Z -3.8333, A 0.000, B 0.000, C 0.000 }
gfCNCPoint3[10121] = {X 476.6273, Y 11.4857, Z -3.8333, A 0.000, B 0.000, C 0.000 }
gfCNCPoint3[10122] = {X 477.8424, Y 10.4985, Z -3.8333, A 0.000, B 0.000, C 0.000 }
gfCNCPoint3[10123] = {X 479.1802, Y 9.6853, Z -3.8333, A 0.000, B 0.000, C 0.000 }
gfCNCPoint3[10124] = {X 480.6160, Y 9.0612, Z -3.8333, A 0.000, B 0.000, C 0.000 }
gfCNCPoint3[10125] = {X 482.1233, Y 8.6378, Z -3.8333, A 0.000, B 0.000, C 0.000 }
gfCNCPoint3[10126] = {X 484.1898, Y 8.3158, Z -3.8333, A 0.000, B 0.000, C 0.000 }
gfCNCPoint3[10127] = {X 486.2782, Y 8.2031, Z -3.8333, A 0.000, B 0.000, C 0.000 }
gfCNCPoint3[10128] = {X 486.9707, Y 8.1909, Z -3.8333, A 0.000, B 0.000, C 0.000 }
gfCNCPoint3[10129] = {X 492.3835, Y 8.1909, Z -3.8333, A 0.000, B 0.000, C 0.000 }
gfCNCPoint3[10130] = {X 492.3835, Y 4.1109, Z -3.8333, A 0.000, B 0.000, C 0.000 }
gfCNCPoint3[10131] = {X 492.3835, Y 4.1109, Z -0.8333, A 0.000, B 0.000, C 0.000 }
gfCNCPoint3[10132] = {X 492.3835, Y 4.1109, Z 11.0000, A 0.000, B 0.000, C 0.000 }
gfCNCPoint3[10133] = {X 533.9639, Y 3.7907, Z 11.0000, A 0.000, B 0.000, C 0.000 }
gfCNCPoint3[10134] = {X 533.9639, Y 3.7907, Z -0.8333, A 0.000, B 0.000, C 0.000 }
gfCNCPoint3[10135] = {X 533.9639, Y 3.7907, Z -3.8333, A 0.000, B 0.000, C 0.000 }
gfCNCPoint3[10136] = {X 533.9638, Y 7.8707, Z -3.8333, A 0.000, B 0.000, C 0.000 }
gfCNCPoint3[10137] = {X 543.7499, Y 7.8709, Z -3.8333, A 0.000, B 0.000, C 0.000 }
gfCNCPoint3[10138] = {X 544.7301, Y 7.9564, Z -3.8333, A 0.000, B 0.000, C 0.000 }
gfCNCPoint3[10139] = {X 545.6656, Y 8.2613, Z -3.8333, A 0.000, B 0.000, C 0.000 }
gfCNCPoint3[10140] = {X 546.5079, Y 8.7697, Z -3.8333, A 0.000, B 0.000, C 0.000 }
gfCNCPoint3[10141] = {X 547.2136, Y 9.4553, Z -3.8333, A 0.000, B 0.000, C 0.000 }
gfCNCPoint3[10142] = {X 547.7461, Y 10.2827, Z -3.8333, A 0.000, B 0.000, C 0.000 }
gfCNCPoint3[10143] = {X 548.0777, Y 11.2090, Z -3.8333, A 0.000, B 0.000, C 0.000 }
gfCNCPoint3[10144] = {X 548.1914, Y 12.1863, Z -3.8333, A 0.000, B 0.000, C 0.000 }
gfCNCPoint3[10145] = {X 548.1912, Y 13.0225, Z -3.8333, A 0.000, B 0.000, C 0.000 }
gfCNCPoint3[10146] = {X 548.0827, Y 13.9406, Z -3.8333, A 0.000, B 0.000, C 0.000 }
gfCNCPoint3[10147] = {X 547.7814, Y 14.8146, Z -3.8333, A 0.000, B 0.000, C 0.000 }
gfCNCPoint3[10148] = {X 547.3010, Y 15.6045, Z -3.8333, A 0.000, B 0.000, C 0.000 }
gfCNCPoint3[10149] = {X 546.6635, Y 16.2741, Z -3.8333, A 0.000, B 0.000, C 0.000 }
gfCNCPoint3[10150] = {X 546.6637, Y 40.9135, Z -3.8333, A 0.000, B 0.000, C 0.000 }
gfCNCPoint3[10151] = {X 546.6859, Y 40.9314, Z -3.8333, A 0.000, B 0.000, C 0.000 }
gfCNCPoint3[10152] = {X 547.3158, Y 41.6013, Z -3.8333, A 0.000, B 0.000, C 0.000 }
gfCNCPoint3[10153] = {X 547.7896, Y 42.3894, Z -3.8333, A 0.000, B 0.000, C 0.000 }
gfCNCPoint3[10154] = {X 548.0859, Y 43.2598, Z -3.8333, A 0.000, B 0.000, C 0.000 }
gfCNCPoint3[10155] = {X 548.1913, Y 44.1733, Z -3.8333, A 0.000, B 0.000, C 0.000 }
gfCNCPoint3[10156] = {X 548.1914, Y 45.0005, Z -3.8333, A 0.000, B 0.000, C 0.000 }
gfCNCPoint3[10157] = {X 548.0777, Y 45.9778, Z -3.8333, A 0.000, B 0.000, C 0.000 }
gfCNCPoint3[10158] = {X 547.7461, Y 46.9041, Z -3.8333, A 0.000, B 0.000, C 0.000 }
gfCNCPoint3[10159] = {X 547.2136, Y 47.7315, Z -3.8333, A 0.000, B 0.000, C 0.000 }
gfCNCPoint3[10160] = {X 546.5079, Y 48.4171, Z -3.8333, A 0.000, B 0.000, C 0.000 }
gfCNCPoint3[10161] = {X 545.6656, Y 48.9254, Z -3.8333, A 0.000, B 0.000, C 0.000 }
gfCNCPoint3[10162] = {X 544.7301, Y 49.2302, Z -3.8333, A 0.000, B 0.000, C 0.000 }
gfCNCPoint3[10163] = {X 543.7499, Y 49.3156, Z -3.8333, A 0.000, B 0.000, C 0.000 }
gfCNCPoint3[10164] = {X 524.0450, Y 49.3161, Z -3.8333, A 0.000, B 0.000, C 0.000 }
gfCNCPoint3[10165] = {X 523.4984, Y 49.9500, Z -3.8333, A 0.000, B 0.000, C 0.000 }
gfCNCPoint3[10166] = {X 522.8435, Y 50.4711, Z -3.8333, A 0.000, B 0.000, C 0.000 }
gfCNCPoint3[10167] = {X 522.1030, Y 50.8613, Z -3.8333, A 0.000, B 0.000, C 0.000 }
gfCNCPoint3[10168] = {X 521.3028, Y 51.1068, Z -3.8333, A 0.000, B 0.000, C 0.000 }
gfCNCPoint3[10169] = {X 520.4709, Y 51.1991, Z -3.8333, A 0.000, B 0.000, C 0.000 }
gfCNCPoint3[10170] = {X 519.7998, Y 51.1991, Z -3.8333, A 0.000, B 0.000, C 0.000 }
gfCNCPoint3[10171] = {X 518.8385, Y 51.0908, Z -3.8333, A 0.000, B 0.000, C 0.000 }
gfCNCPoint3[10172] = {X 517.9254, Y 50.7713, Z -3.8333, A 0.000, B 0.000, C 0.000 }
gfCNCPoint3[10173] = {X 517.1063, Y 50.2566, Z -3.8333, A 0.000, B 0.000, C 0.000 }
gfCNCPoint3[10174] = {X 516.4223, Y 49.5726, Z -3.8333, A 0.000, B 0.000, C 0.000 }
gfCNCPoint3[10175] = {X 515.9076, Y 48.7535, Z -3.8333, A 0.000, B 0.000, C 0.000 }
gfCNCPoint3[10176] = {X 515.5881, Y 47.8404, Z -3.8333, A 0.000, B 0.000, C 0.000 }
gfCNCPoint3[10177] = {X 515.4798, Y 46.8791, Z -3.8333, A 0.000, B 0.000, C 0.000 }
gfCNCPoint3[10178] = {X 515.4798, Y 39.9011, Z -3.8333, A 0.000, B 0.000, C 0.000 }
gfCNCPoint3[10179] = {X 515.5869, Y 38.9451, Z -3.8333, A 0.000, B 0.000, C 0.000 }
gfCNCPoint3[10180] = {X 515.9029, Y 38.0365, Z -3.8333, A 0.000, B 0.000, C 0.000 }
gfCNCPoint3[10181] = {X 516.4121, Y 37.2204, Z -3.8333, A 0.000, B 0.000, C 0.000 }
gfCNCPoint3[10182] = {X 517.0893, Y 36.5372, Z -3.8333, A 0.000, B 0.000, C 0.000 }
gfCNCPoint3[10183] = {X 517.9010, Y 36.0208, Z -3.8333, A 0.000, B 0.000, C 0.000 }
gfCNCPoint3[10184] = {X 518.8067, Y 35.6968, Z -3.8333, A 0.000, B 0.000, C 0.000 }
gfCNCPoint3[10185] = {X 519.7617, Y 35.5813, Z -3.8333, A 0.000, B 0.000, C 0.000 }
gfCNCPoint3[10186] = {X 520.5269, Y 35.5815, Z -3.8333, A 0.000, B 0.000, C 0.000 }
gfCNCPoint3[10187] = {X 521.3534, Y 35.6728, Z -3.8333, A 0.000, B 0.000, C 0.000 }
gfCNCPoint3[10188] = {X 522.1471, Y 35.9207, Z -3.8333, A 0.000, B 0.000, C 0.000 }
gfCNCPoint3[10189] = {X 522.8787, Y 36.3161, Z -3.8333, A 0.000, B 0.000, C 0.000 }
gfCNCPoint3[10190] = {X 523.5209, Y 36.8444, Z -3.8333, A 0.000, B 0.000, C 0.000 }
gfCNCPoint3[10191] = {X 524.0500, Y 37.4859, Z -3.8333, A 0.000, B 0.000, C 0.000 }
gfCNCPoint3[10192] = {X 534.6319, Y 37.4864, Z -3.8333, A 0.000, B 0.000, C 0.000 }
gfCNCPoint3[10193] = {X 534.6319, Y 33.9652, Z -3.8333, A 0.000, B 0.000, C 0.000 }
gfCNCPoint3[10194] = {X 530.1089, Y 33.9666, Z -3.8333, A 0.000, B 0.000, C 0.000 }
gfCNCPoint3[10195] = {X 529.5767, Y 34.6105, Z -3.8333, A 0.000, B 0.000, C 0.000 }
gfCNCPoint3[10196] = {X 528.9306, Y 35.1400, Z -3.8333, A 0.000, B 0.000, C 0.000 }
gfCNCPoint3[10197] = {X 528.1945, Y 35.5352, Z -3.8333, A 0.000, B 0.000, C 0.000 }
gfCNCPoint3[10198] = {X 527.3962, Y 35.7814, Z -3.8333, A 0.000, B 0.000, C 0.000 }
gfCNCPoint3[10199] = {X 526.5655, Y 35.8693, Z -3.8333, A 0.000, B 0.000, C 0.000 }
gfCNCPoint3[10200] = {X 525.8868, Y 35.8694, Z -3.8333, A 0.000, B 0.000, C 0.000 }
gfCNCPoint3[10201] = {X 524.9255, Y 35.7611, Z -3.8333, A 0.000, B 0.000, C 0.000 }
gfCNCPoint3[10202] = {X 524.0124, Y 35.4416, Z -3.8333, A 0.000, B 0.000, C 0.000 }
gfCNCPoint3[10203] = {X 523.1933, Y 34.9270, Z -3.8333, A 0.000, B 0.000, C 0.000 }
gfCNCPoint3[10204] = {X 522.5092, Y 34.2429, Z -3.8333, A 0.000, B 0.000, C 0.000 }
gfCNCPoint3[10205] = {X 521.9946, Y 33.4238, Z -3.8333, A 0.000, B 0.000, C 0.000 }
gfCNCPoint3[10206] = {X 521.6751, Y 32.5107, Z -3.8333, A 0.000, B 0.000, C 0.000 }
gfCNCPoint3[10207] = {X 521.5668, Y 31.5495, Z -3.8333, A 0.000, B 0.000, C 0.000 }
gfCNCPoint3[10208] = {X 521.5668, Y 24.5714, Z -3.8333, A 0.000, B 0.000, C 0.000 }
gfCNCPoint3[10209] = {X 521.6739, Y 23.6153, Z -3.8333, A 0.000, B 0.000, C 0.000 }
gfCNCPoint3[10210] = {X 521.9900, Y 22.7066, Z -3.8333, A 0.000, B 0.000, C 0.000 }
gfCNCPoint3[10211] = {X 522.4994, Y 21.8904, Z -3.8333, A 0.000, B 0.000, C 0.000 }
gfCNCPoint3[10212] = {X 523.1768, Y 21.2071, Z -3.8333, A 0.000, B 0.000, C 0.000 }
gfCNCPoint3[10213] = {X 523.9886, Y 20.6908, Z -3.8333, A 0.000, B 0.000, C 0.000 }
gfCNCPoint3[10214] = {X 524.8946, Y 20.3669, Z -3.8333, A 0.000, B 0.000, C 0.000 }
gfCNCPoint3[10215] = {X 525.8498, Y 20.2516, Z -3.8333, A 0.000, B 0.000, C 0.000 }
gfCNCPoint3[10216] = {X 526.5695, Y 20.2516, Z -3.8333, A 0.000, B 0.000, C 0.000 }
gfCNCPoint3[10217] = {X 527.3946, Y 20.3392, Z -3.8333, A 0.000, B 0.000, C 0.000 }
gfCNCPoint3[10218] = {X 528.1877, Y 20.5828, Z -3.8333, A 0.000, B 0.000, C 0.000 }
gfCNCPoint3[10219] = {X 528.9197, Y 20.9736, Z -3.8333, A 0.000, B 0.000, C 0.000 }
gfCNCPoint3[10220] = {X 529.5634, Y 21.4972, Z -3.8333, A 0.000, B 0.000, C 0.000 }
gfCNCPoint3[10221] = {X 530.0952, Y 22.1341, Z -3.8333, A 0.000, B 0.000, C 0.000 }
gfCNCPoint3[10222] = {X 534.6319, Y 22.1344, Z -3.8333, A 0.000, B 0.000, C 0.000 }
gfCNCPoint3[10223] = {X 534.6319, Y 19.7017, Z -3.8333, A 0.000, B 0.000, C 0.000 }
gfCNCPoint3[10224] = {X 524.1923, Y 19.7013, Z -3.8333, A 0.000, B 0.000, C 0.000 }
gfCNCPoint3[10225] = {X 523.6599, Y 20.3460, Z -3.8333, A 0.000, B 0.000, C 0.000 }
gfCNCPoint3[10226] = {X 523.0132, Y 20.8761, Z -3.8333, A 0.000, B 0.000, C 0.000 }
gfCNCPoint3[10227] = {X 522.2766, Y 21.2716, Z -3.8333, A 0.000, B 0.000, C 0.000 }
gfCNCPoint3[10228] = {X 521.4775, Y 21.5179, Z -3.8333, A 0.000, B 0.000, C 0.000 }
gfCNCPoint3[10229] = {X 520.6460, Y 21.6056, Z -3.8333, A 0.000, B 0.000, C 0.000 }
gfCNCPoint3[10230] = {X 519.9691, Y 21.6057, Z -3.8333, A 0.000, B 0.000, C 0.000 }
gfCNCPoint3[10231] = {X 519.0078, Y 21.4974, Z -3.8333, A 0.000, B 0.000, C 0.000 }
gfCNCPoint3[10232] = {X 518.0947, Y 21.1779, Z -3.8333, A 0.000, B 0.000, C 0.000 }
gfCNCPoint3[10233] = {X 517.2756, Y 20.6632, Z -3.8333, A 0.000, B 0.000, C 0.000 }
gfCNCPoint3[10234] = {X 516.5916, Y 19.9792, Z -3.8333, A 0.000, B 0.000, C 0.000 }
gfCNCPoint3[10235] = {X 516.0769, Y 19.1601, Z -3.8333, A 0.000, B 0.000, C 0.000 }
gfCNCPoint3[10236] = {X 515.7574, Y 18.2470, Z -3.8333, A 0.000, B 0.000, C 0.000 }
gfCNCPoint3[10237] = {X 515.6491, Y 17.2857, Z -3.8333, A 0.000, B 0.000, C 0.000 }
gfCNCPoint3[10238] = {X 515.6491, Y 10.3077, Z -3.8333, A 0.000, B 0.000, C 0.000 }
gfCNCPoint3[10239] = {X 515.7562, Y 9.3519, Z -3.8333, A 0.000, B 0.000, C 0.000 }
gfCNCPoint3[10240] = {X 516.0720, Y 8.4435, Z -3.8333, A 0.000, B 0.000, C 0.000 }
gfCNCPoint3[10241] = {X 516.5811, Y 7.6275, Z -3.8333, A 0.000, B 0.000, C 0.000 }
gfCNCPoint3[10242] = {X 517.2580, Y 6.9443, Z -3.8333, A 0.000, B 0.000, C 0.000 }
gfCNCPoint3[10243] = {X 518.0693, Y 6.4278, Z -3.8333, A 0.000, B 0.000, C 0.000 }
gfCNCPoint3[10244] = {X 518.9748, Y 6.1037, Z -3.8333, A 0.000, B 0.000, C 0.000 }
gfCNCPoint3[10245] = {X 519.9296, Y 5.9879, Z -3.8333, A 0.000, B 0.000, C 0.000 }
gfCNCPoint3[10246] = {X 520.6502, Y 5.9879, Z -3.8333, A 0.000, B 0.000, C 0.000 }
gfCNCPoint3[10247] = {X 521.4757, Y 6.0752, Z -3.8333, A 0.000, B 0.000, C 0.000 }
gfCNCPoint3[10248] = {X 522.2692, Y 6.3187, Z -3.8333, A 0.000, B 0.000, C 0.000 }
gfCNCPoint3[10249] = {X 523.0015, Y 6.7095, Z -3.8333, A 0.000, B 0.000, C 0.000 }
gfCNCPoint3[10250] = {X 523.6456, Y 7.2332, Z -3.8333, A 0.000, B 0.000, C 0.000 }
gfCNCPoint3[10251] = {X 524.1776, Y 7.8704, Z -3.8333, A 0.000, B 0.000, C 0.000 }
gfCNCPoint3[10252] = {X 533.9638, Y 7.8707, Z -3.8333, A 0.000, B 0.000, C 0.000 }
gfCNCPoint3[10253] = {X 533.9639, Y 3.8707, Z -3.8333, A 0.000, B 0.000, C 0.000 }
gfCNCPoint3[10254] = {X 533.9638, Y 7.9507, Z -3.8333, A 0.000, B 0.000, C 0.000 }
gfCNCPoint3[10255] = {X 543.7510, Y 7.9509, Z -3.8333, A 0.000, B 0.000, C 0.000 }
gfCNCPoint3[10256] = {X 544.7132, Y 8.0346, Z -3.8333, A 0.000, B 0.000, C 0.000 }
gfCNCPoint3[10257] = {X 545.6316, Y 8.3337, Z -3.8333, A 0.000, B 0.000, C 0.000 }
gfCNCPoint3[10258] = {X 546.4586, Y 8.8326, Z -3.8333, A 0.000, B 0.000, C 0.000 }
gfCNCPoint3[10259] = {X 547.1514, Y 9.5056, Z -3.8333, A 0.000, B 0.000, C 0.000 }
gfCNCPoint3[10260] = {X 547.6742, Y 10.3177, Z -3.8333, A 0.000, B 0.000, C 0.000 }
gfCNCPoint3[10261] = {X 547.9998, Y 11.2270, Z -3.8333, A 0.000, B 0.000, C 0.000 }
gfCNCPoint3[10262] = {X 548.1114, Y 12.1864, Z -3.8333, A 0.000, B 0.000, C 0.000 }
gfCNCPoint3[10263] = {X 548.1112, Y 13.0217, Z -3.8333, A 0.000, B 0.000, C 0.000 }
gfCNCPoint3[10264] = {X 548.0027, Y 13.9318, Z -3.8333, A 0.000, B 0.000, C 0.000 }
gfCNCPoint3[10265] = {X 547.7011, Y 14.7973, Z -3.8333, A 0.000, B 0.000, C 0.000 }
gfCNCPoint3[10266] = {X 547.2206, Y 15.5778, Z -3.8333, A 0.000, B 0.000, C 0.000 }
gfCNCPoint3[10267] = {X 546.5835, Y 16.2368, Z -3.8333, A 0.000, B 0.000, C 0.000 }
gfCNCPoint3[10268] = {X 546.5837, Y 40.9516, Z -3.8333, A 0.000, B 0.000, C 0.000 }
gfCNCPoint3[10269] = {X 546.6346, Y 40.9928, Z -3.8333, A 0.000, B 0.000, C 0.000 }
gfCNCPoint3[10270] = {X 547.2525, Y 41.6503, Z -3.8333, A 0.000, B 0.000, C 0.000 }
gfCNCPoint3[10271] = {X 547.7173, Y 42.4236, Z -3.8333, A 0.000, B 0.000, C 0.000 }
gfCNCPoint3[10272] = {X 548.0079, Y 43.2777, Z -3.8333, A 0.000, B 0.000, C 0.000 }
gfCNCPoint3[10273] = {X 548.1113, Y 44.1740, Z -3.8333, A 0.000, B 0.000, C 0.000 }
gfCNCPoint3[10274] = {X 548.1114, Y 45.0004, Z -3.8333, A 0.000, B 0.000, C 0.000 }
gfCNCPoint3[10275] = {X 547.9998, Y 45.9598, Z -3.8333, A 0.000, B 0.000, C 0.000 }
gfCNCPoint3[10276] = {X 547.6742, Y 46.8690, Z -3.8333, A 0.000, B 0.000, C 0.000 }
gfCNCPoint3[10277] = {X 547.1514, Y 47.6812, Z -3.8333, A 0.000, B 0.000, C 0.000 }
gfCNCPoint3[10278] = {X 546.4586, Y 48.3541, Z -3.8333, A 0.000, B 0.000, C 0.000 }
gfCNCPoint3[10279] = {X 545.6316, Y 48.8530, Z -3.8333, A 0.000, B 0.000, C 0.000 }
gfCNCPoint3[10280] = {X 544.7132, Y 49.1520, Z -3.8333, A 0.000, B 0.000, C 0.000 }
gfCNCPoint3[10281] = {X 543.7510, Y 49.2356, Z -3.8333, A 0.000, B 0.000, C 0.000 }
gfCNCPoint3[10282] = {X 524.0035, Y 49.2361, Z -3.8333, A 0.000, B 0.000, C 0.000 }
gfCNCPoint3[10283] = {X 523.4667, Y 49.8693, Z -3.8333, A 0.000, B 0.000, C 0.000 }
gfCNCPoint3[10284] = {X 522.8206, Y 50.3904, Z -3.8333, A 0.000, B 0.000, C 0.000 }
gfCNCPoint3[10285] = {X 522.0880, Y 50.7809, Z -3.8333, A 0.000, B 0.000, C 0.000 }
gfCNCPoint3[10286] = {X 521.2951, Y 51.0267, Z -3.8333, A 0.000, B 0.000, C 0.000 }
gfCNCPoint3[10287] = {X 520.4702, Y 51.1191, Z -3.8333, A 0.000, B 0.000, C 0.000 }
gfCNCPoint3[10288] = {X 519.7998, Y 51.1191, Z -3.8333, A 0.000, B 0.000, C 0.000 }
gfCNCPoint3[10289] = {X 518.8563, Y 51.0128, Z -3.8333, A 0.000, B 0.000, C 0.000 }
gfCNCPoint3[10290] = {X 517.9601, Y 50.6992, Z -3.8333, A 0.000, B 0.000, C 0.000 }
gfCNCPoint3[10291] = {X 517.1562, Y 50.1941, Z -3.8333, A 0.000, B 0.000, C 0.000 }
gfCNCPoint3[10292] = {X 516.4848, Y 49.5227, Z -3.8333, A 0.000, B 0.000, C 0.000 }
gfCNCPoint3[10293] = {X 515.9797, Y 48.7188, Z -3.8333, A 0.000, B 0.000, C 0.000 }
gfCNCPoint3[10294] = {X 515.6661, Y 47.8226, Z -3.8333, A 0.000, B 0.000, C 0.000 }
gfCNCPoint3[10295] = {X 515.5598, Y 46.8791, Z -3.8333, A 0.000, B 0.000, C 0.000 }
gfCNCPoint3[10296] = {X 515.5598, Y 39.9011, Z -3.8333, A 0.000, B 0.000, C 0.000 }
gfCNCPoint3[10297] = {X 515.6649, Y 38.9628, Z -3.8333, A 0.000, B 0.000, C 0.000 }
gfCNCPoint3[10298] = {X 515.9751, Y 38.0710, Z -3.8333, A 0.000, B 0.000, C 0.000 }
gfCNCPoint3[10299] = {X 516.4749, Y 37.2700, Z -3.8333, A 0.000, B 0.000, C 0.000 }
gfCNCPoint3[10300] = {X 517.1395, Y 36.5995, Z -3.8333, A 0.000, B 0.000, C 0.000 }
gfCNCPoint3[10301] = {X 517.9361, Y 36.0926, Z -3.8333, A 0.000, B 0.000, C 0.000 }
gfCNCPoint3[10302] = {X 518.8251, Y 35.7746, Z -3.8333, A 0.000, B 0.000, C 0.000 }
gfCNCPoint3[10303] = {X 519.7624, Y 35.6613, Z -3.8333, A 0.000, B 0.000, C 0.000 }
gfCNCPoint3[10304] = {X 520.5258, Y 35.6615, Z -3.8333, A 0.000, B 0.000, C 0.000 }
gfCNCPoint3[10305] = {X 521.3453, Y 35.7528, Z -3.8333, A 0.000, B 0.000, C 0.000 }
gfCNCPoint3[10306] = {X 522.1317, Y 36.0010, Z -3.8333, A 0.000, B 0.000, C 0.000 }
gfCNCPoint3[10307] = {X 522.8551, Y 36.3968, Z -3.8333, A 0.000, B 0.000, C 0.000 }
gfCNCPoint3[10308] = {X 523.4882, Y 36.9251, Z -3.8333, A 0.000, B 0.000, C 0.000 }
gfCNCPoint3[10309] = {X 524.0072, Y 37.5659, Z -3.8333, A 0.000, B 0.000, C 0.000 }
gfCNCPoint3[10310] = {X 534.7119, Y 37.5664, Z -3.8333, A 0.000, B 0.000, C 0.000 }
gfCNCPoint3[10311] = {X 534.7119, Y 33.8852, Z -3.8333, A 0.000, B 0.000, C 0.000 }
gfCNCPoint3[10312] = {X 530.0658, Y 33.8848, Z -3.8333, A 0.000, B 0.000, C 0.000 }
gfCNCPoint3[10313] = {X 530.0419, Y 33.9229, Z -3.8333, A 0.000, B 0.000, C 0.000 }
gfCNCPoint3[10314] = {X 529.5195, Y 34.5546, Z -3.8333, A 0.000, B 0.000, C 0.000 }
gfCNCPoint3[10315] = {X 528.8854, Y 35.0740, Z -3.8333, A 0.000, B 0.000, C 0.000 }
gfCNCPoint3[10316] = {X 528.1632, Y 35.4616, Z -3.8333, A 0.000, B 0.000, C 0.000 }
gfCNCPoint3[10317] = {X 527.3799, Y 35.7031, Z -3.8333, A 0.000, B 0.000, C 0.000 }
gfCNCPoint3[10318] = {X 526.5648, Y 35.7893, Z -3.8333, A 0.000, B 0.000, C 0.000 }
gfCNCPoint3[10319] = {X 525.8868, Y 35.7895, Z -3.8333, A 0.000, B 0.000, C 0.000 }
gfCNCPoint3[10320] = {X 524.9433, Y 35.6831, Z -3.8333, A 0.000, B 0.000, C 0.000 }
gfCNCPoint3[10321] = {X 524.0471, Y 35.3696, Z -3.8333, A 0.000, B 0.000, C 0.000 }
gfCNCPoint3[10322] = {X 523.2432, Y 34.8644, Z -3.8333, A 0.000, B 0.000, C 0.000 }
gfCNCPoint3[10323] = {X 522.5718, Y 34.1930, Z -3.8333, A 0.000, B 0.000, C 0.000 }
gfCNCPoint3[10324] = {X 522.0666, Y 33.3891, Z -3.8333, A 0.000, B 0.000, C 0.000 }
gfCNCPoint3[10325] = {X 521.7531, Y 32.4929, Z -3.8333, A 0.000, B 0.000, C 0.000 }
gfCNCPoint3[10326] = {X 521.6468, Y 31.5495, Z -3.8333, A 0.000, B 0.000, C 0.000 }
gfCNCPoint3[10327] = {X 521.6468, Y 24.5714, Z -3.8333, A 0.000, B 0.000, C 0.000 }
gfCNCPoint3[10328] = {X 521.7519, Y 23.6330, Z -3.8333, A 0.000, B 0.000, C 0.000 }
gfCNCPoint3[10329] = {X 522.0622, Y 22.7411, Z -3.8333, A 0.000, B 0.000, C 0.000 }
gfCNCPoint3[10330] = {X 522.5621, Y 21.9400, Z -3.8333, A 0.000, B 0.000, C 0.000 }
gfCNCPoint3[10331] = {X 523.2270, Y 21.2694, Z -3.8333, A 0.000, B 0.000, C 0.000 }
gfCNCPoint3[10332] = {X 524.0238, Y 20.7626, Z -3.8333, A 0.000, B 0.000, C 0.000 }
gfCNCPoint3[10333] = {X 524.9130, Y 20.4448, Z -3.8333, A 0.000, B 0.000, C 0.000 }
gfCNCPoint3[10334] = {X 525.8505, Y 20.3316, Z -3.8333, A 0.000, B 0.000, C 0.000 }
gfCNCPoint3[10335] = {X 526.5687, Y 20.3316, Z -3.8333, A 0.000, B 0.000, C 0.000 }
gfCNCPoint3[10336] = {X 527.3868, Y 20.4192, Z -3.8333, A 0.000, B 0.000, C 0.000 }
gfCNCPoint3[10337] = {X 528.1725, Y 20.6632, Z -3.8333, A 0.000, B 0.000, C 0.000 }
gfCNCPoint3[10338] = {X 528.8964, Y 21.0543, Z -3.8333, A 0.000, B 0.000, C 0.000 }
gfCNCPoint3[10339] = {X 529.5311, Y 21.5778, Z -3.8333, A 0.000, B 0.000, C 0.000 }
gfCNCPoint3[10340] = {X 530.0527, Y 22.2141, Z -3.8333, A 0.000, B 0.000, C 0.000 }
gfCNCPoint3[10341] = {X 534.7119, Y 22.2144, Z -3.8333, A 0.000, B 0.000, C 0.000 }
gfCNCPoint3[10342] = {X 534.7119, Y 19.6217, Z -3.8333, A 0.000, B 0.000, C 0.000 }
gfCNCPoint3[10343] = {X 524.1492, Y 19.6213, Z -3.8333, A 0.000, B 0.000, C 0.000 }
gfCNCPoint3[10344] = {X 524.1260, Y 19.6566, Z -3.8333, A 0.000, B 0.000, C 0.000 }
gfCNCPoint3[10345] = {X 523.6034, Y 20.2893, Z -3.8333, A 0.000, B 0.000, C 0.000 }
gfCNCPoint3[10346] = {X 522.9687, Y 20.8096, Z -3.8333, A 0.000, B 0.000, C 0.000 }
gfCNCPoint3[10347] = {X 522.2457, Y 21.1978, Z -3.8333, A 0.000, B 0.000, C 0.000 }
gfCNCPoint3[10348] = {X 521.4615, Y 21.4395, Z -3.8333, A 0.000, B 0.000, C 0.000 }
gfCNCPoint3[10349] = {X 520.6453, Y 21.5256, Z -3.8333, A 0.000, B 0.000, C 0.000 }
gfCNCPoint3[10350] = {X 519.9691, Y 21.5257, Z -3.8333, A 0.000, B 0.000, C 0.000 }
gfCNCPoint3[10351] = {X 519.0256, Y 21.4194, Z -3.8333, A 0.000, B 0.000, C 0.000 }
gfCNCPoint3[10352] = {X 518.1294, Y 21.1058, Z -3.8333, A 0.000, B 0.000, C 0.000 }
gfCNCPoint3[10353] = {X 517.3255, Y 20.6007, Z -3.8333, A 0.000, B 0.000, C 0.000 }
gfCNCPoint3[10354] = {X 516.6541, Y 19.9293, Z -3.8333, A 0.000, B 0.000, C 0.000 }
gfCNCPoint3[10355] = {X 516.1490, Y 19.1254, Z -3.8333, A 0.000, B 0.000, C 0.000 }
gfCNCPoint3[10356] = {X 515.8354, Y 18.2292, Z -3.8333, A 0.000, B 0.000, C 0.000 }
gfCNCPoint3[10357] = {X 515.7291, Y 17.2857, Z -3.8333, A 0.000, B 0.000, C 0.000 }
gfCNCPoint3[10358] = {X 515.7291, Y 10.3077, Z -3.8333, A 0.000, B 0.000, C 0.000 }
gfCNCPoint3[10359] = {X 515.8342, Y 9.3696, Z -3.8333, A 0.000, B 0.000, C 0.000 }
gfCNCPoint3[10360] = {X 516.1442, Y 8.4780, Z -3.8333, A 0.000, B 0.000, C 0.000 }
gfCNCPoint3[10361] = {X 516.6438, Y 7.6771, Z -3.8333, A 0.000, B 0.000, C 0.000 }
gfCNCPoint3[10362] = {X 517.3082, Y 7.0066, Z -3.8333, A 0.000, B 0.000, C 0.000 }
gfCNCPoint3[10363] = {X 518.1045, Y 6.4997, Z -3.8333, A 0.000, B 0.000, C 0.000 }
gfCNCPoint3[10364] = {X 518.9932, Y 6.1815, Z -3.8333, A 0.000, B 0.000, C 0.000 }
gfCNCPoint3[10365] = {X 519.9303, Y 6.0679, Z -3.8333, A 0.000, B 0.000, C 0.000 }
gfCNCPoint3[10366] = {X 520.6494, Y 6.0679, Z -3.8333, A 0.000, B 0.000, C 0.000 }
gfCNCPoint3[10367] = {X 521.4679, Y 6.1552, Z -3.8333, A 0.000, B 0.000, C 0.000 }
gfCNCPoint3[10368] = {X 522.2540, Y 6.3991, Z -3.8333, A 0.000, B 0.000, C 0.000 }
gfCNCPoint3[10369] = {X 522.9782, Y 6.7902, Z -3.8333, A 0.000, B 0.000, C 0.000 }
gfCNCPoint3[10370] = {X 523.6132, Y 7.3139, Z -3.8333, A 0.000, B 0.000, C 0.000 }
gfCNCPoint3[10371] = {X 524.1351, Y 7.9504, Z -3.8333, A 0.000, B 0.000, C 0.000 }
gfCNCPoint3[10372] = {X 533.9638, Y 7.9507, Z -3.8333, A 0.000, B 0.000, C 0.000 }
gfCNCPoint3[10373] = {X 533.9639, Y 3.9507, Z -3.8333, A 0.000, B 0.000, C 0.000 }
gfCNCPoint3[10374] = {X 533.9637, Y 8.0307, Z -3.8333, A 0.000, B 0.000, C 0.000 }
gfCNCPoint3[10375] = {X 543.7521, Y 8.0309, Z -3.8333, A 0.000, B 0.000, C 0.000 }
gfCNCPoint3[10376] = {X 544.6964, Y 8.1128, Z -3.8333, A 0.000, B 0.000, C 0.000 }
gfCNCPoint3[10377] = {X 545.5976, Y 8.4061, Z -3.8333, A 0.000, B 0.000, C 0.000 }
gfCNCPoint3[10378] = {X 546.4093, Y 8.8956, Z -3.8333, A 0.000, B 0.000, C 0.000 }
gfCNCPoint3[10379] = {X 547.0892, Y 9.5559, Z -3.8333, A 0.000, B 0.000, C 0.000 }
gfCNCPoint3[10380] = {X 547.6023, Y 10.3528, Z -3.8333, A 0.000, B 0.000, C 0.000 }
gfCNCPoint3[10381] = {X 547.9219, Y 11.2451, Z -3.8333, A 0.000, B 0.000, C 0.000 }
gfCNCPoint3[10382] = {X 548.0314, Y 12.1866, Z -3.8333, A 0.000, B 0.000, C 0.000 }
gfCNCPoint3[10383] = {X 548.0312, Y 13.0208, Z -3.8333, A 0.000, B 0.000, C 0.000 }
gfCNCPoint3[10384] = {X 547.9288, Y 13.8965, Z -3.8333, A 0.000, B 0.000, C 0.000 }
gfCNCPoint3[10385] = {X 547.6441, Y 14.7309, Z -3.8333, A 0.000, B 0.000, C 0.000 }
gfCNCPoint3[10386] = {X 547.1900, Y 15.4865, Z -3.8333, A 0.000, B 0.000, C 0.000 }
gfCNCPoint3[10387] = {X 546.5869, Y 16.1295, Z -3.8333, A 0.000, B 0.000, C 0.000 }
gfCNCPoint3[10388] = {X 546.5035, Y 16.1995, Z -3.8333, A 0.000, B 0.000, C 0.000 }
gfCNCPoint3[10389] = {X 546.5037, Y 40.9897, Z -3.8333, A 0.000, B 0.000, C 0.000 }
gfCNCPoint3[10390] = {X 546.5833, Y 41.0543, Z -3.8333, A 0.000, B 0.000, C 0.000 }
gfCNCPoint3[10391] = {X 547.1892, Y 41.6992, Z -3.8333, A 0.000, B 0.000, C 0.000 }
gfCNCPoint3[10392] = {X 547.6450, Y 42.4578, Z -3.8333, A 0.000, B 0.000, C 0.000 }
gfCNCPoint3[10393] = {X 547.9299, Y 43.2955, Z -3.8333, A 0.000, B 0.000, C 0.000 }
gfCNCPoint3[10394] = {X 548.0313, Y 44.1746, Z -3.8333, A 0.000, B 0.000, C 0.000 }
gfCNCPoint3[10395] = {X 548.0314, Y 45.0003, Z -3.8333, A 0.000, B 0.000, C 0.000 }
gfCNCPoint3[10396] = {X 547.9219, Y 45.9417, Z -3.8333, A 0.000, B 0.000, C 0.000 }
gfCNCPoint3[10397] = {X 547.6023, Y 46.8339, Z -3.8333, A 0.000, B 0.000, C 0.000 }
gfCNCPoint3[10398] = {X 547.0892, Y 47.6309, Z -3.8333, A 0.000, B 0.000, C 0.000 }
gfCNCPoint3[10399] = {X 546.4093, Y 48.2911, Z -3.8333, A 0.000, B 0.000, C 0.000 }
gfCNCPoint3[10400] = {X 545.5976, Y 48.7805, Z -3.8333, A 0.000, B 0.000, C 0.000 }
gfCNCPoint3[10401] = {X 544.6963, Y 49.0738, Z -3.8333, A 0.000, B 0.000, C 0.000 }
gfCNCPoint3[10402] = {X 543.7521, Y 49.1556, Z -3.8333, A 0.000, B 0.000, C 0.000 }
gfCNCPoint3[10403] = {X 523.9615, Y 49.1561, Z -3.8333, A 0.000, B 0.000, C 0.000 }
gfCNCPoint3[10404] = {X 523.4347, Y 49.7886, Z -3.8333, A 0.000, B 0.000, C 0.000 }
gfCNCPoint3[10405] = {X 522.7975, Y 50.3097, Z -3.8333, A 0.000, B 0.000, C 0.000 }
gfCNCPoint3[10406] = {X 522.0729, Y 50.7004, Z -3.8333, A 0.000, B 0.000, C 0.000 }
gfCNCPoint3[10407] = {X 521.2874, Y 50.9465, Z -3.8333, A 0.000, B 0.000, C 0.000 }
gfCNCPoint3[10408] = {X 520.4695, Y 51.0391, Z -3.8333, A 0.000, B 0.000, C 0.000 }
gfCNCPoint3[10409] = {X 519.7998, Y 51.0391, Z -3.8333, A 0.000, B 0.000, C 0.000 }
gfCNCPoint3[10410] = {X 518.8741, Y 50.9348, Z -3.8333, A 0.000, B 0.000, C 0.000 }
gfCNCPoint3[10411] = {X 517.9948, Y 50.6272, Z -3.8333, A 0.000, B 0.000, C 0.000 }
gfCNCPoint3[10412] = {X 517.2061, Y 50.1315, Z -3.8333, A 0.000, B 0.000, C 0.000 }
gfCNCPoint3[10413] = {X 516.5474, Y 49.4728, Z -3.8333, A 0.000, B 0.000, C 0.000 }
gfCNCPoint3[10414] = {X 516.0517, Y 48.6841, Z -3.8333, A 0.000, B 0.000, C 0.000 }
gfCNCPoint3[10415] = {X 515.7441, Y 47.8048, Z -3.8333, A 0.000, B 0.000, C 0.000 }
gfCNCPoint3[10416] = {X 515.6398, Y 46.8791, Z -3.8333, A 0.000, B 0.000, C 0.000 }
gfCNCPoint3[10417] = {X 515.6398, Y 39.9011, Z -3.8333, A 0.000, B 0.000, C 0.000 }
gfCNCPoint3[10418] = {X 515.7429, Y 38.9805, Z -3.8333, A 0.000, B 0.000, C 0.000 }
gfCNCPoint3[10419] = {X 516.0472, Y 38.1056, Z -3.8333, A 0.000, B 0.000, C 0.000 }
gfCNCPoint3[10420] = {X 516.5376, Y 37.3197, Z -3.8333, A 0.000, B 0.000, C 0.000 }
gfCNCPoint3[10421] = {X 517.1897, Y 36.6618, Z -3.8333, A 0.000, B 0.000, C 0.000 }
gfCNCPoint3[10422] = {X 517.9713, Y 36.1645, Z -3.8333, A 0.000, B 0.000, C 0.000 }
gfCNCPoint3[10423] = {X 518.8435, Y 35.8525, Z -3.8333, A 0.000, B 0.000, C 0.000 }
gfCNCPoint3[10424] = {X 519.7631, Y 35.7413, Z -3.8333, A 0.000, B 0.000, C 0.000 }
gfCNCPoint3[10425] = {X 520.5247, Y 35.7415, Z -3.8333, A 0.000, B 0.000, C 0.000 }
gfCNCPoint3[10426] = {X 521.3372, Y 35.8329, Z -3.8333, A 0.000, B 0.000, C 0.000 }
gfCNCPoint3[10427] = {X 522.1161, Y 36.0814, Z -3.8333, A 0.000, B 0.000, C 0.000 }
gfCNCPoint3[10428] = {X 522.8313, Y 36.4775, Z -3.8333, A 0.000, B 0.000, C 0.000 }
gfCNCPoint3[10429] = {X 523.4553, Y 37.0058, Z -3.8333, A 0.000, B 0.000, C 0.000 }
gfCNCPoint3[10430] = {X 523.9638, Y 37.6459, Z -3.8333, A 0.000, B 0.000, C 0.000 }
gfCNCPoint3[10431] = {X 534.7919, Y 37.6464, Z -3.8333, A 0.000, B 0.000, C 0.000 }
gfCNCPoint3[10432] = {X 534.7919, Y 33.8053, Z -3.8333, A 0.000, B 0.000, C 0.000 }
gfCNCPoint3[10433] = {X 530.0216, Y 33.8048, Z -3.8333, A 0.000, B 0.000, C 0.000 }
gfCNCPoint3[10434] = {X 529.9749, Y 33.8792, Z -3.8333, A 0.000, B 0.000, C 0.000 }
gfCNCPoint3[10435] = {X 529.4624, Y 34.4986, Z -3.8333, A 0.000, B 0.000, C 0.000 }
gfCNCPoint3[10436] = {X 528.8403, Y 35.0079, Z -3.8333, A 0.000, B 0.000, C 0.000 }
gfCNCPoint3[10437] = {X 528.1319, Y 35.3880, Z -3.8333, A 0.000, B 0.000, C 0.000 }
gfCNCPoint3[10438] = {X 527.3636, Y 35.6248, Z -3.8333, A 0.000, B 0.000, C 0.000 }
gfCNCPoint3[10439] = {X 526.5641, Y 35.7093, Z -3.8333, A 0.000, B 0.000, C 0.000 }
gfCNCPoint3[10440] = {X 525.8868, Y 35.7095, Z -3.8333, A 0.000, B 0.000, C 0.000 }
gfCNCPoint3[10441] = {X 524.9611, Y 35.6052, Z -3.8333, A 0.000, B 0.000, C 0.000 }
gfCNCPoint3[10442] = {X 524.0818, Y 35.2975, Z -3.8333, A 0.000, B 0.000, C 0.000 }
gfCNCPoint3[10443] = {X 523.2930, Y 34.8019, Z -3.8333, A 0.000, B 0.000, C 0.000 }
gfCNCPoint3[10444] = {X 522.6343, Y 34.1432, Z -3.8333, A 0.000, B 0.000, C 0.000 }
gfCNCPoint3[10445] = {X 522.1387, Y 33.3544, Z -3.8333, A 0.000, B 0.000, C 0.000 }
gfCNCPoint3[10446] = {X 521.8311, Y 32.4751, Z -3.8333, A 0.000, B 0.000, C 0.000 }
gfCNCPoint3[10447] = {X 521.7268, Y 31.5495, Z -3.8333, A 0.000, B 0.000, C 0.000 }
gfCNCPoint3[10448] = {X 521.7268, Y 24.5714, Z -3.8333, A 0.000, B 0.000, C 0.000 }
gfCNCPoint3[10449] = {X 521.8299, Y 23.6507, Z -3.8333, A 0.000, B 0.000, C 0.000 }
gfCNCPoint3[10450] = {X 522.1343, Y 22.7756, Z -3.8333, A 0.000, B 0.000, C 0.000 }
gfCNCPoint3[10451] = {X 522.6248, Y 21.9897, Z -3.8333, A 0.000, B 0.000, C 0.000 }
gfCNCPoint3[10452] = {X 523.2772, Y 21.3317, Z -3.8333, A 0.000, B 0.000, C 0.000 }
gfCNCPoint3[10453] = {X 524.0589, Y 20.8345, Z -3.8333, A 0.000, B 0.000, C 0.000 }
gfCNCPoint3[10454] = {X 524.9313, Y 20.5226, Z -3.8333, A 0.000, B 0.000, C 0.000 }
gfCNCPoint3[10455] = {X 525.8511, Y 20.4116, Z -3.8333, A 0.000, B 0.000, C 0.000 }
gfCNCPoint3[10456] = {X 526.5679, Y 20.4116, Z -3.8333, A 0.000, B 0.000, C 0.000 }
gfCNCPoint3[10457] = {X 527.3789, Y 20.4993, Z -3.8333, A 0.000, B 0.000, C 0.000 }
gfCNCPoint3[10458] = {X 528.1572, Y 20.7436, Z -3.8333, A 0.000, B 0.000, C 0.000 }
gfCNCPoint3[10459] = {X 528.8729, Y 21.1350, Z -3.8333, A 0.000, B 0.000, C 0.000 }
gfCNCPoint3[10460] = {X 529.4984, Y 21.6585, Z -3.8333, A 0.000, B 0.000, C 0.000 }
gfCNCPoint3[10461] = {X 530.0097, Y 22.2941, Z -3.8333, A 0.000, B 0.000, C 0.000 }
gfCNCPoint3[10462] = {X 534.7919, Y 22.2944, Z -3.8333, A 0.000, B 0.000, C 0.000 }
gfCNCPoint3[10463] = {X 534.7919, Y 19.5417, Z -3.8333, A 0.000, B 0.000, C 0.000 }
gfCNCPoint3[10464] = {X 524.1050, Y 19.5413, Z -3.8333, A 0.000, B 0.000, C 0.000 }
gfCNCPoint3[10465] = {X 524.0764, Y 19.5868, Z -3.8333, A 0.000, B 0.000, C 0.000 }
gfCNCPoint3[10466] = {X 523.5640, Y 20.2156, Z -3.8333, A 0.000, B 0.000, C 0.000 }
gfCNCPoint3[10467] = {X 522.9392, Y 20.7330, Z -3.8333, A 0.000, B 0.000, C 0.000 }
gfCNCPoint3[10468] = {X 522.2260, Y 21.1193, Z -3.8333, A 0.000, B 0.000, C 0.000 }
gfCNCPoint3[10469] = {X 521.4513, Y 21.3599, Z -3.8333, A 0.000, B 0.000, C 0.000 }
gfCNCPoint3[10470] = {X 520.6447, Y 21.4456, Z -3.8333, A 0.000, B 0.000, C 0.000 }
gfCNCPoint3[10471] = {X 519.9691, Y 21.4457, Z -3.8333, A 0.000, B 0.000, C 0.000 }
gfCNCPoint3[10472] = {X 519.0434, Y 21.3414, Z -3.8333, A 0.000, B 0.000, C 0.000 }
gfCNCPoint3[10473] = {X 518.1641, Y 21.0337, Z -3.8333, A 0.000, B 0.000, C 0.000 }
gfCNCPoint3[10474] = {X 517.3754, Y 20.5381, Z -3.8333, A 0.000, B 0.000, C 0.000 }
gfCNCPoint3[10475] = {X 516.7167, Y 19.8794, Z -3.8333, A 0.000, B 0.000, C 0.000 }
gfCNCPoint3[10476] = {X 516.2211, Y 19.0907, Z -3.8333, A 0.000, B 0.000, C 0.000 }
gfCNCPoint3[10477] = {X 515.9134, Y 18.2114, Z -3.8333, A 0.000, B 0.000, C 0.000 }
gfCNCPoint3[10478] = {X 515.8091, Y 17.2857, Z -3.8333, A 0.000, B 0.000, C 0.000 }
gfCNCPoint3[10479] = {X 515.8091, Y 10.3077, Z -3.8333, A 0.000, B 0.000, C 0.000 }
gfCNCPoint3[10480] = {X 515.9122, Y 9.3873, Z -3.8333, A 0.000, B 0.000, C 0.000 }
gfCNCPoint3[10481] = {X 516.2164, Y 8.5125, Z -3.8333, A 0.000, B 0.000, C 0.000 }
gfCNCPoint3[10482] = {X 516.7065, Y 7.7267, Z -3.8333, A 0.000, B 0.000, C 0.000 }
gfCNCPoint3[10483] = {X 517.3584, Y 7.0689, Z -3.8333, A 0.000, B 0.000, C 0.000 }
gfCNCPoint3[10484] = {X 518.1397, Y 6.5715, Z -3.8333, A 0.000, B 0.000, C 0.000 }
gfCNCPoint3[10485] = {X 519.0117, Y 6.2594, Z -3.8333, A 0.000, B 0.000, C 0.000 }
gfCNCPoint3[10486] = {X 519.9311, Y 6.1479, Z -3.8333, A 0.000, B 0.000, C 0.000 }
gfCNCPoint3[10487] = {X 520.6487, Y 6.1479, Z -3.8333, A 0.000, B 0.000, C 0.000 }
gfCNCPoint3[10488] = {X 521.4600, Y 6.2353, Z -3.8333, A 0.000, B 0.000, C 0.000 }
gfCNCPoint3[10489] = {X 522.2387, Y 6.4795, Z -3.8333, A 0.000, B 0.000, C 0.000 }
gfCNCPoint3[10490] = {X 522.9547, Y 6.8709, Z -3.8333, A 0.000, B 0.000, C 0.000 }
gfCNCPoint3[10491] = {X 523.5806, Y 7.3946, Z -3.8333, A 0.000, B 0.000, C 0.000 }
gfCNCPoint3[10492] = {X 524.0921, Y 8.0304, Z -3.8333, A 0.000, B 0.000, C 0.000 }
gfCNCPoint3[10493] = {X 533.9637, Y 8.0307, Z -3.8333, A 0.000, B 0.000, C 0.000 }
gfCNCPoint3[10494] = {X 533.9638, Y 4.0307, Z -3.8333, A 0.000, B 0.000, C 0.000 }
gfCNCPoint3[10495] = {X 533.9637, Y 8.1107, Z -3.8333, A 0.000, B 0.000, C 0.000 }
gfCNCPoint3[10496] = {X 543.7532, Y 8.1109, Z -3.8333, A 0.000, B 0.000, C 0.000 }
gfCNCPoint3[10497] = {X 544.6795, Y 8.1910, Z -3.8333, A 0.000, B 0.000, C 0.000 }
gfCNCPoint3[10498] = {X 545.5637, Y 8.4786, Z -3.8333, A 0.000, B 0.000, C 0.000 }
gfCNCPoint3[10499] = {X 546.3599, Y 8.9586, Z -3.8333, A 0.000, B 0.000, C 0.000 }
gfCNCPoint3[10500] = {X 547.0270, Y 9.6062, Z -3.8333, A 0.000, B 0.000, C 0.000 }
gfCNCPoint3[10501] = {X 547.5304, Y 10.3879, Z -3.8333, A 0.000, B 0.000, C 0.000 }
gfCNCPoint3[10502] = {X 547.8439, Y 11.2632, Z -3.8333, A 0.000, B 0.000, C 0.000 }
gfCNCPoint3[10503] = {X 547.9514, Y 12.1867, Z -3.8333, A 0.000, B 0.000, C 0.000 }
gfCNCPoint3[10504] = {X 547.9512, Y 13.0200, Z -3.8333, A 0.000, B 0.000, C 0.000 }
gfCNCPoint3[10505] = {X 547.8507, Y 13.8788, Z -3.8333, A 0.000, B 0.000, C 0.000 }
gfCNCPoint3[10506] = {X 547.5716, Y 14.6972, Z -3.8333, A 0.000, B 0.000, C 0.000 }
gfCNCPoint3[10507] = {X 547.1262, Y 15.4383, Z -3.8333, A 0.000, B 0.000, C 0.000 }
gfCNCPoint3[10508] = {X 546.5346, Y 16.0689, Z -3.8333, A 0.000, B 0.000, C 0.000 }
gfCNCPoint3[10509] = {X 546.4800, Y 16.1152, Z -3.8333, A 0.000, B 0.000, C 0.000 }
gfCNCPoint3[10510] = {X 546.4245, Y 16.1605, Z -3.8333, A 0.000, B 0.000, C 0.000 }
gfCNCPoint3[10511] = {X 546.4237, Y 41.0278, Z -3.8333, A 0.000, B 0.000, C 0.000 }
gfCNCPoint3[10512] = {X 546.5320, Y 41.1157, Z -3.8333, A 0.000, B 0.000, C 0.000 }
gfCNCPoint3[10513] = {X 547.1259, Y 41.7482, Z -3.8333, A 0.000, B 0.000, C 0.000 }
gfCNCPoint3[10514] = {X 547.5726, Y 42.4919, Z -3.8333, A 0.000, B 0.000, C 0.000 }
gfCNCPoint3[10515] = {X 547.8520, Y 43.3134, Z -3.8333, A 0.000, B 0.000, C 0.000 }
gfCNCPoint3[10516] = {X 547.9513, Y 44.1753, Z -3.8333, A 0.000, B 0.000, C 0.000 }
gfCNCPoint3[10517] = {X 547.9514, Y 45.0001, Z -3.8333, A 0.000, B 0.000, C 0.000 }
gfCNCPoint3[10518] = {X 547.8439, Y 45.9236, Z -3.8333, A 0.000, B 0.000, C 0.000 }
gfCNCPoint3[10519] = {X 547.5304, Y 46.7989, Z -3.8333, A 0.000, B 0.000, C 0.000 }
gfCNCPoint3[10520] = {X 547.0270, Y 47.5805, Z -3.8333, A 0.000, B 0.000, C 0.000 }
gfCNCPoint3[10521] = {X 546.3599, Y 48.2281, Z -3.8333, A 0.000, B 0.000, C 0.000 }
gfCNCPoint3[10522] = {X 545.5637, Y 48.7081, Z -3.8333, A 0.000, B 0.000, C 0.000 }
gfCNCPoint3[10523] = {X 544.6795, Y 48.9955, Z -3.8333, A 0.000, B 0.000, C 0.000 }
gfCNCPoint3[10524] = {X 543.7532, Y 49.0756, Z -3.8333, A 0.000, B 0.000, C 0.000 }
gfCNCPoint3[10525] = {X 523.9190, Y 49.0761, Z -3.8333, A 0.000, B 0.000, C 0.000 }
gfCNCPoint3[10526] = {X 523.4023, Y 49.7079, Z -3.8333, A 0.000, B 0.000, C 0.000 }
gfCNCPoint3[10527] = {X 522.7742, Y 50.2290, Z -3.8333, A 0.000, B 0.000, C 0.000 }
gfCNCPoint3[10528] = {X 522.0577, Y 50.6200, Z -3.8333, A 0.000, B 0.000, C 0.000 }
gfCNCPoint3[10529] = {X 521.2797, Y 50.8664, Z -3.8333, A 0.000, B 0.000, C 0.000 }
gfCNCPoint3[10530] = {X 520.4688, Y 50.9591, Z -3.8333, A 0.000, B 0.000, C 0.000 }
gfCNCPoint3[10531] = {X 519.7998, Y 50.9591, Z -3.8333, A 0.000, B 0.000, C 0.000 }
gfCNCPoint3[10532] = {X 518.8919, Y 50.8568, Z -3.8333, A 0.000, B 0.000, C 0.000 }
gfCNCPoint3[10533] = {X 518.0295, Y 50.5551, Z -3.8333, A 0.000, B 0.000, C 0.000 }
gfCNCPoint3[10534] = {X 517.2559, Y 50.0690, Z -3.8333, A 0.000, B 0.000, C 0.000 }
gfCNCPoint3[10535] = {X 516.6099, Y 49.4230, Z -3.8333, A 0.000, B 0.000, C 0.000 }
gfCNCPoint3[10536] = {X 516.1238, Y 48.6494, Z -3.8333, A 0.000, B 0.000, C 0.000 }
gfCNCPoint3[10537] = {X 515.8221, Y 47.7870, Z -3.8333, A 0.000, B 0.000, C 0.000 }
gfCNCPoint3[10538] = {X 515.7198, Y 46.8791, Z -3.8333, A 0.000, B 0.000, C 0.000 }
gfCNCPoint3[10539] = {X 515.7198, Y 39.9011, Z -3.8333, A 0.000, B 0.000, C 0.000 }
gfCNCPoint3[10540] = {X 515.8209, Y 38.9982, Z -3.8333, A 0.000, B 0.000, C 0.000 }
gfCNCPoint3[10541] = {X 516.1194, Y 38.1401, Z -3.8333, A 0.000, B 0.000, C 0.000 }
gfCNCPoint3[10542] = {X 516.6003, Y 37.3693, Z -3.8333, A 0.000, B 0.000, C 0.000 }
gfCNCPoint3[10543] = {X 517.2399, Y 36.7241, Z -3.8333, A 0.000, B 0.000, C 0.000 }
gfCNCPoint3[10544] = {X 518.0064, Y 36.2364, Z -3.8333, A 0.000, B 0.000, C 0.000 }
gfCNCPoint3[10545] = {X 518.8619, Y 35.9304, Z -3.8333, A 0.000, B 0.000, C 0.000 }
gfCNCPoint3[10546] = {X 519.7638, Y 35.8213, Z -3.8333, A 0.000, B 0.000, C 0.000 }
gfCNCPoint3[10547] = {X 520.5236, Y 35.8215, Z -3.8333, A 0.000, B 0.000, C 0.000 }
gfCNCPoint3[10548] = {X 521.3289, Y 35.9129, Z -3.8333, A 0.000, B 0.000, C 0.000 }
gfCNCPoint3[10549] = {X 522.1003, Y 36.1618, Z -3.8333, A 0.000, B 0.000, C 0.000 }
gfCNCPoint3[10550] = {X 522.8073, Y 36.5582, Z -3.8333, A 0.000, B 0.000, C 0.000 }
gfCNCPoint3[10551] = {X 523.4219, Y 37.0865, Z -3.8333, A 0.000, B 0.000, C 0.000 }
gfCNCPoint3[10552] = {X 523.9200, Y 37.7259, Z -3.8333, A 0.000, B 0.000, C 0.000 }
gfCNCPoint3[10553] = {X 534.8719, Y 37.7264, Z -3.8333, A 0.000, B 0.000, C 0.000 }
gfCNCPoint3[10554] = {X 534.8719, Y 33.7253, Z -3.8333, A 0.000, B 0.000, C 0.000 }
gfCNCPoint3[10555] = {X 529.9774, Y 33.7248, Z -3.8333, A 0.000, B 0.000, C 0.000 }
gfCNCPoint3[10556] = {X 529.9071, Y 33.8366, Z -3.8333, A 0.000, B 0.000, C 0.000 }
gfCNCPoint3[10557] = {X 529.2612, Y 34.5790, Z -3.8333, A 0.000, B 0.000, C 0.000 }
gfCNCPoint3[10558] = {X 528.4563, Y 35.1452, Z -3.8333, A 0.000, B 0.000, C 0.000 }
gfCNCPoint3[10559] = {X 527.5392, Y 35.5023, Z -3.8333, A 0.000, B 0.000, C 0.000 }
gfCNCPoint3[10560] = {X 526.5634, Y 35.6293, Z -3.8333, A 0.000, B 0.000, C 0.000 }
gfCNCPoint3[10561] = {X 525.8868, Y 35.6295, Z -3.8333, A 0.000, B 0.000, C 0.000 }
gfCNCPoint3[10562] = {X 524.9789, Y 35.5272, Z -3.8333, A 0.000, B 0.000, C 0.000 }
gfCNCPoint3[10563] = {X 524.1165, Y 35.2254, Z -3.8333, A 0.000, B 0.000, C 0.000 }
gfCNCPoint3[10564] = {X 523.3429, Y 34.7393, Z -3.8333, A 0.000, B 0.000, C 0.000 }
gfCNCPoint3[10565] = {X 522.6969, Y 34.0933, Z -3.8333, A 0.000, B 0.000, C 0.000 }
gfCNCPoint3[10566] = {X 522.2108, Y 33.3197, Z -3.8333, A 0.000, B 0.000, C 0.000 }
gfCNCPoint3[10567] = {X 521.9091, Y 32.4573, Z -3.8333, A 0.000, B 0.000, C 0.000 }
gfCNCPoint3[10568] = {X 521.8068, Y 31.5495, Z -3.8333, A 0.000, B 0.000, C 0.000 }
gfCNCPoint3[10569] = {X 521.8068, Y 24.5714, Z -3.8333, A 0.000, B 0.000, C 0.000 }
gfCNCPoint3[10570] = {X 521.9079, Y 23.6684, Z -3.8333, A 0.000, B 0.000, C 0.000 }
gfCNCPoint3[10571] = {X 522.2065, Y 22.8102, Z -3.8333, A 0.000, B 0.000, C 0.000 }
gfCNCPoint3[10572] = {X 522.6876, Y 22.0393, Z -3.8333, A 0.000, B 0.000, C 0.000 }
gfCNCPoint3[10573] = {X 523.3273, Y 21.3940, Z -3.8333, A 0.000, B 0.000, C 0.000 }
gfCNCPoint3[10574] = {X 524.0941, Y 20.9064, Z -3.8333, A 0.000, B 0.000, C 0.000 }
gfCNCPoint3[10575] = {X 524.9497, Y 20.6005, Z -3.8333, A 0.000, B 0.000, C 0.000 }
gfCNCPoint3[10576] = {X 525.8518, Y 20.4916, Z -3.8333, A 0.000, B 0.000, C 0.000 }
gfCNCPoint3[10577] = {X 526.5672, Y 20.4916, Z -3.8333, A 0.000, B 0.000, C 0.000 }
gfCNCPoint3[10578] = {X 527.3710, Y 20.5794, Z -3.8333, A 0.000, B 0.000, C 0.000 }
gfCNCPoint3[10579] = {X 528.1417, Y 20.8239, Z -3.8333, A 0.000, B 0.000, C 0.000 }
gfCNCPoint3[10580] = {X 528.8491, Y 21.2157, Z -3.8333, A 0.000, B 0.000, C 0.000 }
gfCNCPoint3[10581] = {X 529.4653, Y 21.7393, Z -3.8333, A 0.000, B 0.000, C 0.000 }
gfCNCPoint3[10582] = {X 529.9662, Y 22.3741, Z -3.8333, A 0.000, B 0.000, C 0.000 }
gfCNCPoint3[10583] = {X 534.8719, Y 22.3744, Z -3.8333, A 0.000, B 0.000, C 0.000 }
gfCNCPoint3[10584] = {X 534.8719, Y 19.4617, Z -3.8333, A 0.000, B 0.000, C 0.000 }
gfCNCPoint3[10585] = {X 524.0608, Y 19.4613, Z -3.8333, A 0.000, B 0.000, C 0.000 }
gfCNCPoint3[10586] = {X 524.0087, Y 19.5442, Z -3.8333, A 0.000, B 0.000, C 0.000 }
gfCNCPoint3[10587] = {X 523.5061, Y 20.1604, Z -3.8333, A 0.000, B 0.000, C 0.000 }
gfCNCPoint3[10588] = {X 522.8935, Y 20.6674, Z -3.8333, A 0.000, B 0.000, C 0.000 }
gfCNCPoint3[10589] = {X 522.1942, Y 21.0459, Z -3.8333, A 0.000, B 0.000, C 0.000 }
gfCNCPoint3[10590] = {X 521.4348, Y 21.2816, Z -3.8333, A 0.000, B 0.000, C 0.000 }
gfCNCPoint3[10591] = {X 520.6440, Y 21.3656, Z -3.8333, A 0.000, B 0.000, C 0.000 }
gfCNCPoint3[10592] = {X 519.9691, Y 21.3657, Z -3.8333, A 0.000, B 0.000, C 0.000 }
gfCNCPoint3[10593] = {X 519.0612, Y 21.2634, Z -3.8333, A 0.000, B 0.000, C 0.000 }
gfCNCPoint3[10594] = {X 518.1989, Y 20.9617, Z -3.8333, A 0.000, B 0.000, C 0.000 }
gfCNCPoint3[10595] = {X 517.4253, Y 20.4756, Z -3.8333, A 0.000, B 0.000, C 0.000 }
gfCNCPoint3[10596] = {X 516.7792, Y 19.8296, Z -3.8333, A 0.000, B 0.000, C 0.000 }
gfCNCPoint3[10597] = {X 516.2932, Y 19.0560, Z -3.8333, A 0.000, B 0.000, C 0.000 }
gfCNCPoint3[10598] = {X 515.9914, Y 18.1936, Z -3.8333, A 0.000, B 0.000, C 0.000 }
gfCNCPoint3[10599] = {X 515.8891, Y 17.2857, Z -3.8333, A 0.000, B 0.000, C 0.000 }
gfCNCPoint3[10600] = {X 515.8891, Y 10.3077, Z -3.8333, A 0.000, B 0.000, C 0.000 }
gfCNCPoint3[10601] = {X 515.9902, Y 9.4050, Z -3.8333, A 0.000, B 0.000, C 0.000 }
gfCNCPoint3[10602] = {X 516.2885, Y 8.5471, Z -3.8333, A 0.000, B 0.000, C 0.000 }
gfCNCPoint3[10603] = {X 516.7693, Y 7.7764, Z -3.8333, A 0.000, B 0.000, C 0.000 }
gfCNCPoint3[10604] = {X 517.4086, Y 7.1312, Z -3.8333, A 0.000, B 0.000, C 0.000 }
gfCNCPoint3[10605] = {X 518.1749, Y 6.6434, Z -3.8333, A 0.000, B 0.000, C 0.000 }
gfCNCPoint3[10606] = {X 519.0301, Y 6.3372, Z -3.8333, A 0.000, B 0.000, C 0.000 }
gfCNCPoint3[10607] = {X 519.9318, Y 6.2279, Z -3.8333, A 0.000, B 0.000, C 0.000 }
gfCNCPoint3[10608] = {X 520.6480, Y 6.2279, Z -3.8333, A 0.000, B 0.000, C 0.000 }
gfCNCPoint3[10609] = {X 521.4522, Y 6.3154, Z -3.8333, A 0.000, B 0.000, C 0.000 }
gfCNCPoint3[10610] = {X 522.2233, Y 6.5599, Z -3.8333, A 0.000, B 0.000, C 0.000 }
gfCNCPoint3[10611] = {X 522.9310, Y 6.9516, Z -3.8333, A 0.000, B 0.000, C 0.000 }
gfCNCPoint3[10612] = {X 523.5475, Y 7.4754, Z -3.8333, A 0.000, B 0.000, C 0.000 }
gfCNCPoint3[10613] = {X 524.0486, Y 8.1104, Z -3.8333, A 0.000, B 0.000, C 0.000 }
gfCNCPoint3[10614] = {X 533.9637, Y 8.1107, Z -3.8333, A 0.000, B 0.000, C 0.000 }
gfCNCPoint3[10615] = {X 533.9638, Y 4.1107, Z -3.8333, A 0.000, B 0.000, C 0.000 }
gfCNCPoint3[10616] = {X 533.9637, Y 8.1907, Z -3.8333, A 0.000, B 0.000, C 0.000 }
gfCNCPoint3[10617] = {X 543.7544, Y 8.1909, Z -3.8333, A 0.000, B 0.000, C 0.000 }
gfCNCPoint3[10618] = {X 544.6627, Y 8.2693, Z -3.8333, A 0.000, B 0.000, C 0.000 }
gfCNCPoint3[10619] = {X 545.5297, Y 8.5510, Z -3.8333, A 0.000, B 0.000, C 0.000 }
gfCNCPoint3[10620] = {X 546.3106, Y 9.0216, Z -3.8333, A 0.000, B 0.000, C 0.000 }
gfCNCPoint3[10621] = {X 546.9648, Y 9.6565, Z -3.8333, A 0.000, B 0.000, C 0.000 }
gfCNCPoint3[10622] = {X 547.4585, Y 10.4230, Z -3.8333, A 0.000, B 0.000, C 0.000 }
gfCNCPoint3[10623] = {X 547.7660, Y 11.2813, Z -3.8333, A 0.000, B 0.000, C 0.000 }
gfCNCPoint3[10624] = {X 547.8714, Y 12.1869, Z -3.8333, A 0.000, B 0.000, C 0.000 }
gfCNCPoint3[10625] = {X 547.8712, Y 13.0192, Z -3.8333, A 0.000, B 0.000, C 0.000 }
gfCNCPoint3[10626] = {X 547.7727, Y 13.8612, Z -3.8333, A 0.000, B 0.000, C 0.000 }
gfCNCPoint3[10627] = {X 547.4990, Y 14.6635, Z -3.8333, A 0.000, B 0.000, C 0.000 }
gfCNCPoint3[10628] = {X 547.0624, Y 15.3901, Z -3.8333, A 0.000, B 0.000, C 0.000 }
gfCNCPoint3[10629] = {X 546.4824, Y 16.0083, Z -3.8333, A 0.000, B 0.000, C 0.000 }
gfCNCPoint3[10630] = {X 546.4147, Y 16.0654, Z -3.8333, A 0.000, B 0.000, C 0.000 }
gfCNCPoint3[10631] = {X 546.3458, Y 16.1209, Z -3.8333, A 0.000, B 0.000, C 0.000 }
gfCNCPoint3[10632] = {X 546.3435, Y 16.3114, Z -3.8333, A 0.000, B 0.000, C 0.000 }
gfCNCPoint3[10633] = {X 546.3437, Y 41.0659, Z -3.8333, A 0.000, B 0.000, C 0.000 }
gfCNCPoint3[10634] = {X 546.4826, Y 41.1787, Z -3.8333, A 0.000, B 0.000, C 0.000 }
gfCNCPoint3[10635] = {X 547.0687, Y 41.8052, Z -3.8333, A 0.000, B 0.000, C 0.000 }
gfCNCPoint3[10636] = {X 547.5077, Y 42.5422, Z -3.8333, A 0.000, B 0.000, C 0.000 }
gfCNCPoint3[10637] = {X 547.7795, Y 43.3559, Z -3.8333, A 0.000, B 0.000, C 0.000 }
gfCNCPoint3[10638] = {X 547.8714, Y 44.2089, Z -3.8333, A 0.000, B 0.000, C 0.000 }
gfCNCPoint3[10639] = {X 547.8714, Y 45.0000, Z -3.8333, A 0.000, B 0.000, C 0.000 }
gfCNCPoint3[10640] = {X 547.7660, Y 45.9055, Z -3.8333, A 0.000, B 0.000, C 0.000 }
gfCNCPoint3[10641] = {X 547.4585, Y 46.7638, Z -3.8333, A 0.000, B 0.000, C 0.000 }
gfCNCPoint3[10642] = {X 546.9648, Y 47.5302, Z -3.8333, A 0.000, B 0.000, C 0.000 }
gfCNCPoint3[10643] = {X 546.3106, Y 48.1651, Z -3.8333, A 0.000, B 0.000, C 0.000 }
gfCNCPoint3[10644] = {X 545.5297, Y 48.6356, Z -3.8333, A 0.000, B 0.000, C 0.000 }
gfCNCPoint3[10645] = {X 544.6627, Y 48.9173, Z -3.8333, A 0.000, B 0.000, C 0.000 }
gfCNCPoint3[10646] = {X 543.7544, Y 48.9956, Z -3.8333, A 0.000, B 0.000, C 0.000 }
gfCNCPoint3[10647] = {X 523.8759, Y 48.9961, Z -3.8333, A 0.000, B 0.000, C 0.000 }
gfCNCPoint3[10648] = {X 523.3696, Y 49.6271, Z -3.8333, A 0.000, B 0.000, C 0.000 }
gfCNCPoint3[10649] = {X 522.7506, Y 50.1482, Z -3.8333, A 0.000, B 0.000, C 0.000 }
gfCNCPoint3[10650] = {X 522.0424, Y 50.5395, Z -3.8333, A 0.000, B 0.000, C 0.000 }
gfCNCPoint3[10651] = {X 521.2719, Y 50.7863, Z -3.8333, A 0.000, B 0.000, C 0.000 }
gfCNCPoint3[10652] = {X 520.4681, Y 50.8791, Z -3.8333, A 0.000, B 0.000, C 0.000 }
gfCNCPoint3[10653] = {X 519.7998, Y 50.8791, Z -3.8333, A 0.000, B 0.000, C 0.000 }
gfCNCPoint3[10654] = {X 518.9097, Y 50.7788, Z -3.8333, A 0.000, B 0.000, C 0.000 }
gfCNCPoint3[10655] = {X 518.0642, Y 50.4830, Z -3.8333, A 0.000, B 0.000, C 0.000 }
gfCNCPoint3[10656] = {X 517.3058, Y 50.0064, Z -3.8333, A 0.000, B 0.000, C 0.000 }
gfCNCPoint3[10657] = {X 516.6724, Y 49.3731, Z -3.8333, A 0.000, B 0.000, C 0.000 }
gfCNCPoint3[10658] = {X 516.1959, Y 48.6147, Z -3.8333, A 0.000, B 0.000, C 0.000 }
gfCNCPoint3[10659] = {X 515.9001, Y 47.7692, Z -3.8333, A 0.000, B 0.000, C 0.000 }
gfCNCPoint3[10660] = {X 515.7998, Y 46.8791, Z -3.8333, A 0.000, B 0.000, C 0.000 }
gfCNCPoint3[10661] = {X 515.7998, Y 39.9011, Z -3.8333, A 0.000, B 0.000, C 0.000 }
gfCNCPoint3[10662] = {X 515.9001, Y 39.0110, Z -3.8333, A 0.000, B 0.000, C 0.000 }
gfCNCPoint3[10663] = {X 516.1959, Y 38.1655, Z -3.8333, A 0.000, B 0.000, C 0.000 }
gfCNCPoint3[10664] = {X 516.6725, Y 37.4071, Z -3.8333, A 0.000, B 0.000, C 0.000 }
gfCNCPoint3[10665] = {X 517.3058, Y 36.7737, Z -3.8333, A 0.000, B 0.000, C 0.000 }
gfCNCPoint3[10666] = {X 518.0643, Y 36.2972, Z -3.8333, A 0.000, B 0.000, C 0.000 }
gfCNCPoint3[10667] = {X 518.9098, Y 36.0014, Z -3.8333, A 0.000, B 0.000, C 0.000 }
gfCNCPoint3[10668] = {X 519.7998, Y 35.9011, Z -3.8333, A 0.000, B 0.000, C 0.000 }
gfCNCPoint3[10669] = {X 520.5225, Y 35.9015, Z -3.8333, A 0.000, B 0.000, C 0.000 }
gfCNCPoint3[10670] = {X 521.3207, Y 35.9930, Z -3.8333, A 0.000, B 0.000, C 0.000 }
gfCNCPoint3[10671] = {X 522.0844, Y 36.2422, Z -3.8333, A 0.000, B 0.000, C 0.000 }
gfCNCPoint3[10672] = {X 522.7830, Y 36.6389, Z -3.8333, A 0.000, B 0.000, C 0.000 }
gfCNCPoint3[10673] = {X 523.3881, Y 37.1673, Z -3.8333, A 0.000, B 0.000, C 0.000 }
gfCNCPoint3[10674] = {X 523.8755, Y 37.8059, Z -3.8333, A 0.000, B 0.000, C 0.000 }
gfCNCPoint3[10675] = {X 534.9519, Y 37.8064, Z -3.8333, A 0.000, B 0.000, C 0.000 }
gfCNCPoint3[10676] = {X 534.9519, Y 34.0452, Z -3.8333, A 0.000, B 0.000, C 0.000 }
gfCNCPoint3[10677] = {X 534.9526, Y 33.6453, Z -3.8333, A 0.000, B 0.000, C 0.000 }
gfCNCPoint3[10678] = {X 529.9332, Y 33.6448, Z -3.8333, A 0.000, B 0.000, C 0.000 }
gfCNCPoint3[10679] = {X 529.8229, Y 33.8180, Z -3.8333, A 0.000, B 0.000, C 0.000 }
gfCNCPoint3[10680] = {X 529.1834, Y 34.5413, Z -3.8333, A 0.000, B 0.000, C 0.000 }
gfCNCPoint3[10681] = {X 528.3893, Y 35.0903, Z -3.8333, A 0.000, B 0.000, C 0.000 }
gfCNCPoint3[10682] = {X 527.4867, Y 35.4330, Z -3.8333, A 0.000, B 0.000, C 0.000 }
gfCNCPoint3[10683] = {X 526.5283, Y 35.5495, Z -3.8333, A 0.000, B 0.000, C 0.000 }
gfCNCPoint3[10684] = {X 525.8868, Y 35.5495, Z -3.8333, A 0.000, B 0.000, C 0.000 }
gfCNCPoint3[10685] = {X 524.9967, Y 35.4492, Z -3.8333, A 0.000, B 0.000, C 0.000 }
gfCNCPoint3[10686] = {X 524.1512, Y 35.1533, Z -3.8333, A 0.000, B 0.000, C 0.000 }
gfCNCPoint3[10687] = {X 523.3928, Y 34.6768, Z -3.8333, A 0.000, B 0.000, C 0.000 }
gfCNCPoint3[10688] = {X 522.7594, Y 34.0434, Z -3.8333, A 0.000, B 0.000, C 0.000 }
gfCNCPoint3[10689] = {X 522.2829, Y 33.2850, Z -3.8333, A 0.000, B 0.000, C 0.000 }
gfCNCPoint3[10690] = {X 521.9870, Y 32.4395, Z -3.8333, A 0.000, B 0.000, C 0.000 }
gfCNCPoint3[10691] = {X 521.8868, Y 31.5495, Z -3.8333, A 0.000, B 0.000, C 0.000 }
gfCNCPoint3[10692] = {X 521.8868, Y 24.5714, Z -3.8333, A 0.000, B 0.000, C 0.000 }
gfCNCPoint3[10693] = {X 521.9870, Y 23.6813, Z -3.8333, A 0.000, B 0.000, C 0.000 }
gfCNCPoint3[10694] = {X 522.2829, Y 22.8359, Z -3.8333, A 0.000, B 0.000, C 0.000 }
gfCNCPoint3[10695] = {X 522.7594, Y 22.0775, Z -3.8333, A 0.000, B 0.000, C 0.000 }
gfCNCPoint3[10696] = {X 523.3928, Y 21.4441, Z -3.8333, A 0.000, B 0.000, C 0.000 }
gfCNCPoint3[10697] = {X 524.1512, Y 20.9675, Z -3.8333, A 0.000, B 0.000, C 0.000 }
gfCNCPoint3[10698] = {X 524.9967, Y 20.6717, Z -3.8333, A 0.000, B 0.000, C 0.000 }
gfCNCPoint3[10699] = {X 525.8868, Y 20.5714, Z -3.8333, A 0.000, B 0.000, C 0.000 }
gfCNCPoint3[10700] = {X 526.5664, Y 20.5716, Z -3.8333, A 0.000, B 0.000, C 0.000 }
gfCNCPoint3[10701] = {X 527.3630, Y 20.6595, Z -3.8333, A 0.000, B 0.000, C 0.000 }
gfCNCPoint3[10702] = {X 528.1261, Y 20.9044, Z -3.8333, A 0.000, B 0.000, C 0.000 }
gfCNCPoint3[10703] = {X 528.8251, Y 21.2965, Z -3.8333, A 0.000, B 0.000, C 0.000 }
gfCNCPoint3[10704] = {X 529.4319, Y 21.8201, Z -3.8333, A 0.000, B 0.000, C 0.000 }
gfCNCPoint3[10705] = {X 529.9221, Y 22.4541, Z -3.8333, A 0.000, B 0.000, C 0.000 }
gfCNCPoint3[10706] = {X 534.9519, Y 22.4544, Z -3.8333, A 0.000, B 0.000, C 0.000 }
gfCNCPoint3[10707] = {X 534.9519, Y 19.7816, Z -3.8333, A 0.000, B 0.000, C 0.000 }
gfCNCPoint3[10708] = {X 534.9527, Y 19.3817, Z -3.8333, A 0.000, B 0.000, C 0.000 }
gfCNCPoint3[10709] = {X 524.0166, Y 19.3813, Z -3.8333, A 0.000, B 0.000, C 0.000 }
gfCNCPoint3[10710] = {X 523.9052, Y 19.5544, Z -3.8333, A 0.000, B 0.000, C 0.000 }
gfCNCPoint3[10711] = {X 523.2657, Y 20.2776, Z -3.8333, A 0.000, B 0.000, C 0.000 }
gfCNCPoint3[10712] = {X 522.4715, Y 20.8266, Z -3.8333, A 0.000, B 0.000, C 0.000 }
gfCNCPoint3[10713] = {X 521.5690, Y 21.1692, Z -3.8333, A 0.000, B 0.000, C 0.000 }
gfCNCPoint3[10714] = {X 520.6107, Y 21.2857, Z -3.8333, A 0.000, B 0.000, C 0.000 }
gfCNCPoint3[10715] = {X 519.9691, Y 21.2857, Z -3.8333, A 0.000, B 0.000, C 0.000 }
gfCNCPoint3[10716] = {X 519.0790, Y 21.1854, Z -3.8333, A 0.000, B 0.000, C 0.000 }
gfCNCPoint3[10717] = {X 518.2336, Y 20.8896, Z -3.8333, A 0.000, B 0.000, C 0.000 }
gfCNCPoint3[10718] = {X 517.4751, Y 20.4130, Z -3.8333, A 0.000, B 0.000, C 0.000 }
gfCNCPoint3[10719] = {X 516.8418, Y 19.7797, Z -3.8333, A 0.000, B 0.000, C 0.000 }
gfCNCPoint3[10720] = {X 516.3652, Y 19.0212, Z -3.8333, A 0.000, B 0.000, C 0.000 }
gfCNCPoint3[10721] = {X 516.0694, Y 18.1758, Z -3.8333, A 0.000, B 0.000, C 0.000 }
gfCNCPoint3[10722] = {X 515.9691, Y 17.2857, Z -3.8333, A 0.000, B 0.000, C 0.000 }
gfCNCPoint3[10723] = {X 515.9691, Y 10.3077, Z -3.8333, A 0.000, B 0.000, C 0.000 }
gfCNCPoint3[10724] = {X 516.0694, Y 9.4176, Z -3.8333, A 0.000, B 0.000, C 0.000 }
gfCNCPoint3[10725] = {X 516.3652, Y 8.5721, Z -3.8333, A 0.000, B 0.000, C 0.000 }
gfCNCPoint3[10726] = {X 516.8418, Y 7.8137, Z -3.8333, A 0.000, B 0.000, C 0.000 }
gfCNCPoint3[10727] = {X 517.4752, Y 7.1803, Z -3.8333, A 0.000, B 0.000, C 0.000 }
gfCNCPoint3[10728] = {X 518.2336, Y 6.7038, Z -3.8333, A 0.000, B 0.000, C 0.000 }
gfCNCPoint3[10729] = {X 519.0791, Y 6.4080, Z -3.8333, A 0.000, B 0.000, C 0.000 }
gfCNCPoint3[10730] = {X 519.9692, Y 6.3077, Z -3.8333, A 0.000, B 0.000, C 0.000 }
gfCNCPoint3[10731] = {X 520.6472, Y 6.3079, Z -3.8333, A 0.000, B 0.000, C 0.000 }
gfCNCPoint3[10732] = {X 521.4442, Y 6.3955, Z -3.8333, A 0.000, B 0.000, C 0.000 }
gfCNCPoint3[10733] = {X 522.2077, Y 6.6403, Z -3.8333, A 0.000, B 0.000, C 0.000 }
gfCNCPoint3[10734] = {X 522.9070, Y 7.0324, Z -3.8333, A 0.000, B 0.000, C 0.000 }
gfCNCPoint3[10735] = {X 523.5140, Y 7.5561, Z -3.8333, A 0.000, B 0.000, C 0.000 }
gfCNCPoint3[10736] = {X 524.0045, Y 8.1904, Z -3.8333, A 0.000, B 0.000, C 0.000 }
gfCNCPoint3[10737] = {X 533.9637, Y 8.1907, Z -3.8333, A 0.000, B 0.000, C 0.000 }
gfCNCPoint3[10738] = {X 533.9638, Y 4.1107, Z -3.8333, A 0.000, B 0.000, C 0.000 }
gfCNCPoint3[10739] = {X 533.9638, Y 4.1107, Z -0.8333, A 0.000, B 0.000, C 0.000 }
gfCNCPoint3[10740] = {X 533.9638, Y 4.1107, Z 11.0000, A 0.000, B 0.000, C 0.000 }
gfCNCPoint3[10741] = {X 419.6139, Y 26.5283, Z 11.0000, A 0.000, B 0.000, C 0.000 }
gfCNCPoint3[10742] = {X 419.6139, Y 26.5283, Z -0.8333, A 0.000, B 0.000, C 0.000 }
gfCNCPoint3[10743] = {X 419.6139, Y 26.5283, Z -3.8333, A 0.000, B 0.000, C 0.000 }
gfCNCPoint3[10744] = {X 416.1504, Y 24.3717, Z -3.8333, A 0.000, B 0.000, C 0.000 }
gfCNCPoint3[10745] = {X 411.5466, Y 31.7650, Z -3.8333, A 0.000, B 0.000, C 0.000 }
gfCNCPoint3[10746] = {X 411.5473, Y 40.8981, Z -3.8333, A 0.000, B 0.000, C 0.000 }
gfCNCPoint3[10747] = {X 412.1854, Y 41.5839, Z -3.8333, A 0.000, B 0.000, C 0.000 }
gfCNCPoint3[10748] = {X 412.6656, Y 42.3883, Z -3.8333, A 0.000, B 0.000, C 0.000 }
gfCNCPoint3[10749] = {X 412.9665, Y 43.2755, Z -3.8333, A 0.000, B 0.000, C 0.000 }
gfCNCPoint3[10750] = {X 413.0747, Y 44.2060, Z -3.8333, A 0.000, B 0.000, C 0.000 }
gfCNCPoint3[10751] = {X 413.0747, Y 45.0002, Z -3.8333, A 0.000, B 0.000, C 0.000 }
gfCNCPoint3[10752] = {X 412.9663, Y 45.9614, Z -3.8333, A 0.000, B 0.000, C 0.000 }
gfCNCPoint3[10753] = {X 412.6468, Y 46.8745, Z -3.8333, A 0.000, B 0.000, C 0.000 }
gfCNCPoint3[10754] = {X 412.1321, Y 47.6935, Z -3.8333, A 0.000, B 0.000, C 0.000 }
gfCNCPoint3[10755] = {X 411.4481, Y 48.3776, Z -3.8333, A 0.000, B 0.000, C 0.000 }
gfCNCPoint3[10756] = {X 410.6290, Y 48.8922, Z -3.8333, A 0.000, B 0.000, C 0.000 }
gfCNCPoint3[10757] = {X 409.7159, Y 49.2117, Z -3.8333, A 0.000, B 0.000, C 0.000 }
gfCNCPoint3[10758] = {X 408.7547, Y 49.3200, Z -3.8333, A 0.000, B 0.000, C 0.000 }
gfCNCPoint3[10759] = {X 402.3112, Y 49.3200, Z -3.8333, A 0.000, B 0.000, C 0.000 }
gfCNCPoint3[10760] = {X 401.3546, Y 49.2127, Z -3.8333, A 0.000, B 0.000, C 0.000 }
gfCNCPoint3[10761] = {X 400.4455, Y 48.8963, Z -3.8333, A 0.000, B 0.000, C 0.000 }
gfCNCPoint3[10762] = {X 399.6290, Y 48.3864, Z -3.8333, A 0.000, B 0.000, C 0.000 }
gfCNCPoint3[10763] = {X 398.9457, Y 47.7084, Z -3.8333, A 0.000, B 0.000, C 0.000 }
gfCNCPoint3[10764] = {X 398.4295, Y 46.8959, Z -3.8333, A 0.000, B 0.000, C 0.000 }
gfCNCPoint3[10765] = {X 398.1060, Y 45.9892, Z -3.8333, A 0.000, B 0.000, C 0.000 }
gfCNCPoint3[10766] = {X 397.9913, Y 45.0335, Z -3.8333, A 0.000, B 0.000, C 0.000 }
gfCNCPoint3[10767] = {X 397.9916, Y 44.1528, Z -3.8333, A 0.000, B 0.000, C 0.000 }
gfCNCPoint3[10768] = {X 398.1015, Y 43.2391, Z -3.8333, A 0.000, B 0.000, C 0.000 }
gfCNCPoint3[10769] = {X 398.4024, Y 42.3694, Z -3.8333, A 0.000, B 0.000, C 0.000 }
gfCNCPoint3[10770] = {X 398.8807, Y 41.5832, Z -3.8333, A 0.000, B 0.000, C 0.000 }
gfCNCPoint3[10771] = {X 399.5147, Y 40.9161, Z -3.8333, A 0.000, B 0.000, C 0.000 }
gfCNCPoint3[10772] = {X 399.4729, Y 31.5997, Z -3.8333, A 0.000, B 0.000, C 0.000 }
gfCNCPoint3[10773] = {X 393.5129, Y 21.2357, Z -3.8333, A 0.000, B 0.000, C 0.000 }
gfCNCPoint3[10774] = {X 392.6261, Y 19.7272, Z -3.8333, A 0.000, B 0.000, C 0.000 }
gfCNCPoint3[10775] = {X 391.7105, Y 18.2359, Z -3.8333, A 0.000, B 0.000, C 0.000 }
gfCNCPoint3[10776] = {X 391.2293, Y 17.5673, Z -3.8333, A 0.000, B 0.000, C 0.000 }
gfCNCPoint3[10777] = {X 390.6671, Y 16.9653, Z -3.8333, A 0.000, B 0.000, C 0.000 }
gfCNCPoint3[10778] = {X 389.7903, Y 16.4729, Z -3.8333, A 0.000, B 0.000, C 0.000 }
gfCNCPoint3[10779] = {X 389.0511, Y 15.7912, Z -3.8333, A 0.000, B 0.000, C 0.000 }
gfCNCPoint3[10780] = {X 388.4896, Y 14.9570, Z -3.8333, A 0.000, B 0.000, C 0.000 }
gfCNCPoint3[10781] = {X 388.1361, Y 14.0156, Z -3.8333, A 0.000, B 0.000, C 0.000 }
gfCNCPoint3[10782] = {X 388.0098, Y 13.0180, Z -3.8333, A 0.000, B 0.000, C 0.000 }
gfCNCPoint3[10783] = {X 388.0096, Y 12.1868, Z -3.8333, A 0.000, B 0.000, C 0.000 }
gfCNCPoint3[10784] = {X 388.1179, Y 11.2255, Z -3.8333, A 0.000, B 0.000, C 0.000 }
gfCNCPoint3[10785] = {X 388.4374, Y 10.3125, Z -3.8333, A 0.000, B 0.000, C 0.000 }
gfCNCPoint3[10786] = {X 388.9521, Y 9.4933, Z -3.8333, A 0.000, B 0.000, C 0.000 }
gfCNCPoint3[10787] = {X 389.6361, Y 8.8093, Z -3.8333, A 0.000, B 0.000, C 0.000 }
gfCNCPoint3[10788] = {X 390.4552, Y 8.2946, Z -3.8333, A 0.000, B 0.000, C 0.000 }
gfCNCPoint3[10789] = {X 391.3683, Y 7.9751, Z -3.8333, A 0.000, B 0.000, C 0.000 }
gfCNCPoint3[10790] = {X 392.3296, Y 7.8668, Z -3.8333, A 0.000, B 0.000, C 0.000 }
gfCNCPoint3[10791] = {X 399.1118, Y 7.8668, Z -3.8333, A 0.000, B 0.000, C 0.000 }
gfCNCPoint3[10792] = {X 400.0730, Y 7.9751, Z -3.8333, A 0.000, B 0.000, C 0.000 }
gfCNCPoint3[10793] = {X 400.9861, Y 8.2946, Z -3.8333, A 0.000, B 0.000, C 0.000 }
gfCNCPoint3[10794] = {X 401.8052, Y 8.8093, Z -3.8333, A 0.000, B 0.000, C 0.000 }
gfCNCPoint3[10795] = {X 402.4893, Y 9.4933, Z -3.8333, A 0.000, B 0.000, C 0.000 }
gfCNCPoint3[10796] = {X 403.0039, Y 10.3124, Z -3.8333, A 0.000, B 0.000, C 0.000 }
gfCNCPoint3[10797] = {X 403.3234, Y 11.2255, Z -3.8333, A 0.000, B 0.000, C 0.000 }
gfCNCPoint3[10798] = {X 403.4318, Y 12.1868, Z -3.8333, A 0.000, B 0.000, C 0.000 }
gfCNCPoint3[10799] = {X 403.4318, Y 12.9781, Z -3.8333, A 0.000, B 0.000, C 0.000 }
gfCNCPoint3[10800] = {X 403.3293, Y 13.9134, Z -3.8333, A 0.000, B 0.000, C 0.000 }
gfCNCPoint3[10801] = {X 403.0267, Y 14.8043, Z -3.8333, A 0.000, B 0.000, C 0.000 }
gfCNCPoint3[10802] = {X 405.3566, Y 18.8233, Z -3.8333, A 0.000, B 0.000, C 0.000 }
gfCNCPoint3[10803] = {X 407.8735, Y 14.7540, Z -3.8333, A 0.000, B 0.000, C 0.000 }
gfCNCPoint3[10804] = {X 407.5920, Y 13.9045, Z -3.8333, A 0.000, B 0.000, C 0.000 }
gfCNCPoint3[10805] = {X 407.4917, Y 13.0151, Z -3.8333, A 0.000, B 0.000, C 0.000 }
gfCNCPoint3[10806] = {X 407.4915, Y 12.1868, Z -3.8333, A 0.000, B 0.000, C 0.000 }
gfCNCPoint3[10807] = {X 407.5999, Y 11.2255, Z -3.8333, A 0.000, B 0.000, C 0.000 }
gfCNCPoint3[10808] = {X 407.9194, Y 10.3124, Z -3.8333, A 0.000, B 0.000, C 0.000 }
gfCNCPoint3[10809] = {X 408.4340, Y 9.4933, Z -3.8333, A 0.000, B 0.000, C 0.000 }
gfCNCPoint3[10810] = {X 409.1181, Y 8.8093, Z -3.8333, A 0.000, B 0.000, C 0.000 }
gfCNCPoint3[10811] = {X 409.9372, Y 8.2946, Z -3.8333, A 0.000, B 0.000, C 0.000 }
gfCNCPoint3[10812] = {X 410.8502, Y 7.9751, Z -3.8333, A 0.000, B 0.000, C 0.000 }
gfCNCPoint3[10813] = {X 411.8115, Y 7.8668, Z -3.8333, A 0.000, B 0.000, C 0.000 }
gfCNCPoint3[10814] = {X 419.3245, Y 7.8668, Z -3.8333, A 0.000, B 0.000, C 0.000 }
gfCNCPoint3[10815] = {X 420.2858, Y 7.9751, Z -3.8333, A 0.000, B 0.000, C 0.000 }
gfCNCPoint3[10816] = {X 421.1988, Y 8.2946, Z -3.8333, A 0.000, B 0.000, C 0.000 }
gfCNCPoint3[10817] = {X 422.0179, Y 8.8093, Z -3.8333, A 0.000, B 0.000, C 0.000 }
gfCNCPoint3[10818] = {X 422.7020, Y 9.4933, Z -3.8333, A 0.000, B 0.000, C 0.000 }
gfCNCPoint3[10819] = {X 423.2166, Y 10.3124, Z -3.8333, A 0.000, B 0.000, C 0.000 }
gfCNCPoint3[10820] = {X 423.5361, Y 11.2255, Z -3.8333, A 0.000, B 0.000, C 0.000 }
gfCNCPoint3[10821] = {X 423.6445, Y 12.1868, Z -3.8333, A 0.000, B 0.000, C 0.000 }
gfCNCPoint3[10822] = {X 423.6445, Y 12.9804, Z -3.8333, A 0.000, B 0.000, C 0.000 }
gfCNCPoint3[10823] = {X 423.5513, Y 13.8469, Z -3.8333, A 0.000, B 0.000, C 0.000 }
gfCNCPoint3[10824] = {X 423.2887, Y 14.6779, Z -3.8333, A 0.000, B 0.000, C 0.000 }
gfCNCPoint3[10825] = {X 422.8669, Y 15.4405, Z -3.8333, A 0.000, B 0.000, C 0.000 }
gfCNCPoint3[10826] = {X 422.3027, Y 16.1047, Z -3.8333, A 0.000, B 0.000, C 0.000 }
gfCNCPoint3[10827] = {X 421.6182, Y 16.6441, Z -3.8333, A 0.000, B 0.000, C 0.000 }
gfCNCPoint3[10828] = {X 420.8406, Y 17.0375, Z -3.8333, A 0.000, B 0.000, C 0.000 }
gfCNCPoint3[10829] = {X 420.1242, Y 18.0010, Z -3.8333, A 0.000, B 0.000, C 0.000 }
gfCNCPoint3[10830] = {X 419.4759, Y 19.0115, Z -3.8333, A 0.000, B 0.000, C 0.000 }
gfCNCPoint3[10831] = {X 417.9942, Y 21.4107, Z -3.8333, A 0.000, B 0.000, C 0.000 }
gfCNCPoint3[10832] = {X 416.1504, Y 24.3717, Z -3.8333, A 0.000, B 0.000, C 0.000 }
gfCNCPoint3[10833] = {X 419.5459, Y 26.4860, Z -3.8333, A 0.000, B 0.000, C 0.000 }
gfCNCPoint3[10834] = {X 416.0825, Y 24.3294, Z -3.8333, A 0.000, B 0.000, C 0.000 }
gfCNCPoint3[10835] = {X 411.4666, Y 31.7422, Z -3.8333, A 0.000, B 0.000, C 0.000 }
gfCNCPoint3[10836] = {X 411.4673, Y 40.9348, Z -3.8333, A 0.000, B 0.000, C 0.000 }
gfCNCPoint3[10837] = {X 412.1050, Y 41.6102, Z -3.8333, A 0.000, B 0.000, C 0.000 }
gfCNCPoint3[10838] = {X 412.5853, Y 42.4054, Z -3.8333, A 0.000, B 0.000, C 0.000 }
gfCNCPoint3[10839] = {X 412.8864, Y 43.2842, Z -3.8333, A 0.000, B 0.000, C 0.000 }
gfCNCPoint3[10840] = {X 412.9947, Y 44.2068, Z -3.8333, A 0.000, B 0.000, C 0.000 }
gfCNCPoint3[10841] = {X 412.9947, Y 45.0002, Z -3.8333, A 0.000, B 0.000, C 0.000 }
gfCNCPoint3[10842] = {X 412.8883, Y 45.9436, Z -3.8333, A 0.000, B 0.000, C 0.000 }
gfCNCPoint3[10843] = {X 412.5747, Y 46.8398, Z -3.8333, A 0.000, B 0.000, C 0.000 }
gfCNCPoint3[10844] = {X 412.0696, Y 47.6437, Z -3.8333, A 0.000, B 0.000, C 0.000 }
gfCNCPoint3[10845] = {X 411.3982, Y 48.3150, Z -3.8333, A 0.000, B 0.000, C 0.000 }
gfCNCPoint3[10846] = {X 410.5943, Y 48.8201, Z -3.8333, A 0.000, B 0.000, C 0.000 }
gfCNCPoint3[10847] = {X 409.6981, Y 49.1337, Z -3.8333, A 0.000, B 0.000, C 0.000 }
gfCNCPoint3[10848] = {X 408.7547, Y 49.2400, Z -3.8333, A 0.000, B 0.000, C 0.000 }
gfCNCPoint3[10849] = {X 402.3112, Y 49.2400, Z -3.8333, A 0.000, B 0.000, C 0.000 }
gfCNCPoint3[10850] = {X 401.3723, Y 49.1347, Z -3.8333, A 0.000, B 0.000, C 0.000 }
gfCNCPoint3[10851] = {X 400.4800, Y 48.8242, Z -3.8333, A 0.000, B 0.000, C 0.000 }
gfCNCPoint3[10852] = {X 399.6786, Y 48.3237, Z -3.8333, A 0.000, B 0.000, C 0.000 }
gfCNCPoint3[10853] = {X 399.0080, Y 47.6582, Z -3.8333, A 0.000, B 0.000, C 0.000 }
gfCNCPoint3[10854] = {X 398.5013, Y 46.8608, Z -3.8333, A 0.000, B 0.000, C 0.000 }
gfCNCPoint3[10855] = {X 398.1839, Y 45.9709, Z -3.8333, A 0.000, B 0.000, C 0.000 }
gfCNCPoint3[10856] = {X 398.0713, Y 45.0329, Z -3.8333, A 0.000, B 0.000, C 0.000 }
gfCNCPoint3[10857] = {X 398.0716, Y 44.1538, Z -3.8333, A 0.000, B 0.000, C 0.000 }
gfCNCPoint3[10858] = {X 398.1815, Y 43.2480, Z -3.8333, A 0.000, B 0.000, C 0.000 }
gfCNCPoint3[10859] = {X 398.4827, Y 42.3867, Z -3.8333, A 0.000, B 0.000, C 0.000 }
gfCNCPoint3[10860] = {X 398.9612, Y 41.6098, Z -3.8333, A 0.000, B 0.000, C 0.000 }
gfCNCPoint3[10861] = {X 399.5948, Y 40.9532, Z -3.8333, A 0.000, B 0.000, C 0.000 }
gfCNCPoint3[10862] = {X 399.5528, Y 31.5782, Z -3.8333, A 0.000, B 0.000, C 0.000 }
gfCNCPoint3[10863] = {X 393.5823, Y 21.1958, Z -3.8333, A 0.000, B 0.000, C 0.000 }
gfCNCPoint3[10864] = {X 392.6947, Y 19.6860, Z -3.8333, A 0.000, B 0.000, C 0.000 }
gfCNCPoint3[10865] = {X 391.7783, Y 18.1934, Z -3.8333, A 0.000, B 0.000, C 0.000 }
gfCNCPoint3[10866] = {X 391.2865, Y 17.5109, Z -3.8333, A 0.000, B 0.000, C 0.000 }
gfCNCPoint3[10867] = {X 390.7112, Y 16.8970, Z -3.8333, A 0.000, B 0.000, C 0.000 }
gfCNCPoint3[10868] = {X 389.8467, Y 16.4150, Z -3.8333, A 0.000, B 0.000, C 0.000 }
gfCNCPoint3[10869] = {X 389.1175, Y 15.7457, Z -3.8333, A 0.000, B 0.000, C 0.000 }
gfCNCPoint3[10870] = {X 388.5634, Y 14.9255, Z -3.8333, A 0.000, B 0.000, C 0.000 }
gfCNCPoint3[10871] = {X 388.2144, Y 13.9992, Z -3.8333, A 0.000, B 0.000, C 0.000 }
gfCNCPoint3[10872] = {X 388.0898, Y 13.0173, Z -3.8333, A 0.000, B 0.000, C 0.000 }
gfCNCPoint3[10873] = {X 388.0896, Y 12.1868, Z -3.8333, A 0.000, B 0.000, C 0.000 }
